// Run Station(s) (define when each needs to run)
fbStationINHeatAndSteam(
	aVehiclesStationFIFO:= aVehiclesStationFIFO,
	stReservation:= fbTrack.P_stReservation,
	stModeStateIn:= Input.Station.Station1.ModeState, 
	stModeStateOut := Output.Station.Station1.ModeState,
	bVehicleReadyAtInput:= eSeq <> E_VehicleOnStation.Idle, 
	bVehicleReadyAtOutput:= , 
	nCellStateCmd:= DINT_TO_UINT(eCommand),
	stJobDataIn:= Input.Station.Station1.JobData,  
	stConfigIn:= Input.Station.Station1.CurrentConfiguration, 
	stUpcomingConfigIn:= Input.Station.Station1.UpcomingConfiguration, 
	stControlIn := Input.Station.Station1.Control,
	stAdditionalDataIn := Input.Station.Station1.AdditionalData,
	sDistanceInDevice := Input.Transport.Configuration.Stations[2].StationLocation1.Position - Input.Transport.Configuration.Stations[1].StationLocation1.Position,
	stVehicleDataStaion := fbTrack.P_stVehicleDataOnStation,
	stJobDataOut := Output.Station.Station1.JobData,  
	stOEE := Output.Station.Station1.OEE, 
	stErrorWarning := Output.Station.Station1.ErrorWarning, 
	stConfigOut := Output.Station.Station1.CurrentConfiguration,
	stUpcomingConfigOut := Output.Station.Station1.UpcomingConfiguration,
	stOperationalDataOut := Output.Station.Station1.OperationalData, 
	stSustainabilityData := Output.Station.Station1.SustainabilityData, 
	stAdditionalDataOut := Output.Station.Station1.AdditionalData 	);
	
fbStationOUTHeatAndSteam(
	stModeStateIn:= Input.Station.Station2.ModeState, 
	stModeStateOut := Output.Station.Station2.ModeState,
	bVehicleReadyAtInput:= , 
	bVehicleReadyAtOutput:= , 
	nCellStateCmd:= DINT_TO_UINT(eCommand),
	stJobDataIn:= Input.Station.Station2.JobData,  
	stConfigIn:= Input.Station.Station2.CurrentConfiguration, 
	stUpcomingConfigIn:= Input.Station.Station2.UpcomingConfiguration, 
	stControlIn := Input.Station.Station2.Control,
	stAdditionalDataIn := Input.Station.Station1.AdditionalData,
	stJobDataOut := Output.Station.Station2.JobData,  
	stOEE := Output.Station.Station2.OEE, 
	stErrorWarning := Output.Station.Station2.ErrorWarning, 
	stConfigOut := Output.Station.Station2.CurrentConfiguration,
	stUpcomingConfigOut := Output.Station.Station2.UpcomingConfiguration,
	stOperationalDataOut := Output.Station.Station2.OperationalData, 
	stSustainabilityData := Output.Station.Station2.SustainabilityData, 
	stAdditionalDataOut := Output.Station.Station2.AdditionalData 	);

	
// Run Track Client
fbTrack(bEnable := , // Enabled in State Resetting
		bEStopOK := TRUE,
		bSuspend := , 
		bReset:= , 
		stCommand:= Input.Transport.Command,
		stMappingIn:= input.Transport.Mapping,
		stAdditionalDataIn:= Input.Transport.AdditionalData,
		bConnectedMethod=> , 
		bBusyMethod=> , 
		bConnectedNode=> , 
		bErrorMethod=> , 
		nErrorMethodID=> , 
		bErrorNode=> , 
		nErrorNodeID=> , 
		stStatus := Output.Transport.Status,
		stMappingOut := Output.Transport.Mapping, 
		stAdditionaldataOut := Output.Transport.AdditionalData,
		bStarted=> , 
		bSuspended=> 	);


//Set Station ready for vehicle to track
fbTrack.P_StationEmptyReady := eSeq = E_VehicleOnStation.Idle;
//fbTrack.P_bStationReady:=fbStationINHeatAndSteam.bStationReadyIn;

//Vehicles on station FIFO handling
M_VehicleOnStation(iCarrierCount=>diVehiclesInDevice);


//Set station empty for track - for vehicles going straight through
fbTrack.P_bStationEmpty:= diVehiclesInDevice = 0;

//Set FIFO for Station IN and Track Client
//fbStationINHeatAndSteam.P_CarriersFIFO := aVehiclesStationFIFO;
fbTrack.P_CarriersFIFO := aVehiclesStationFIFO;
END_METHOD

METHOD PROTECTED M_ErrorWarning
VAR_INPUT
END_VAR
VAR
	iAlNo				: UINT;
	iNoOfAlarms			: UINT;
	iNoOfWarnings		: UINT;
	bST1ErrWarDataChange: BOOL;
	bST2ErrWarDataChange: BOOL;
	bCellDataChange		: BOOL;
	bTCErrWarDataChange	: BOOL;
END_VAR
//Alarm / Warnings Cell
//bCellDataChange S= 
//M_ErrorWarningObj(arErrorWaringData:= arErrorWarningDataCell,
//	bActive:= eLineCtrl_EStop <> E_TwinSAFE_Logic_State.RUN, 
//	iErrorWarningType:= 2, 
//	diErrorWarningID:= E_AlarmCategory.Safety + 0, 
//	sDeviceID:= 'Global Safety',
//	iSeverity:= 2, 
//	iNativeID:= 0, 
//	sNativeMessage:= 'Emergency stop Line Controller');

//bCellDataChange S= 
//M_ErrorWarningObj(arErrorWaringData:= arErrorWarningDataCell,
//	bActive:= NOT bEStop_OK, 
//	iErrorWarningType:= 2, 
//	diErrorWarningID:= E_AlarmCategory.Safety + 20, 
//	sDeviceID:= 'Local Safety',
//	iSeverity:= 2, 
//	iNativeID:= 0, 
//	sNativeMessage:= 'Emergency stop Cell');

//bCellDataChange S= 
//M_ErrorWarningObj(arErrorWaringData:= arErrorWarningDataCell,
//	bActive:= eSHL_F70 <> E_TwinSAFE_Logic_State.RUN, 
//	iErrorWarningType:= 2, 
//	diErrorWarningID:= E_AlarmCategory.Safety + 21, 
//	sDeviceID:= 'Local Safety',
//	iSeverity:= 2, 
//	iNativeID:= 0, 
//	sNativeMessage:= 'Emergency stop Robot');
	
//bCellDataChange S= 
//M_ErrorWarningObj(arErrorWaringData:= arErrorWarningDataCell,
//	bActive:= NOT bDoor_OK, 
//	iErrorWarningType:= 2, 
//	diErrorWarningID:= E_AlarmCategory.Safety + 22, 
//	sDeviceID:= 'Local Safety',
//	iSeverity:= 2, 
//	iNativeID:= 0, 
//	sNativeMessage:= 'Cell Door 1 Not OK');
	
//bCellDataChange S= 
//M_ErrorWarningObj(arErrorWaringData:= arErrorWarningDataCell,
//	bActive:= stStatusData.e03_11_AK01_M3011 = E_Cylinder_Sta.Cyl_Sta_Err, 
//	iErrorWarningType:= 2, 
//	diErrorWarningID:= E_AlarmCategory.LifterStation1Device + 0, 
//	sDeviceID:= 'Lifter Station 1',
//	iSeverity:= 2, 
//	iNativeID:= 0, 
//	sNativeMessage:= 'Error Radial Gripper');
	
//bCellDataChange S= 
//M_ErrorWarningObj(arErrorWaringData:= arErrorWarningDataCell,
//	bActive:= stStatusData.e03_11_AK01_M3015 = E_Cylinder_Sta.Cyl_Sta_Err, 
//	iErrorWarningType:= 2, 
//	diErrorWarningID:= E_AlarmCategory.LifterStation1Device + 1, 
//	sDeviceID:= 'Lifter Station 1',
//	iSeverity:= 2, 
//	iNativeID:= 0, 
//	sNativeMessage:= 'Error Lifter Cylinder');
	
//bCellDataChange S= 
//M_ErrorWarningObj(arErrorWaringData:= arErrorWarningDataCell,
//	bActive:= stStatusData.e03_11_AK01_M3111 = E_Cylinder_Sta.Cyl_Sta_Err, 
//	iErrorWarningType:= 2, 
//	diErrorWarningID:= E_AlarmCategory.LifterStation2Device + 0, 
//	sDeviceID:= 'Lifter Station 2',
//	iSeverity:= 2, 
//	iNativeID:= 0, 
//	sNativeMessage:= 'Error Radial Gripper');
	
//bCellDataChange S= 
//M_ErrorWarningObj(arErrorWaringData:= arErrorWarningDataCell,
//	bActive:= stStatusData.e03_11_AK01_M3115 = E_Cylinder_Sta.Cyl_Sta_Err, 
//	iErrorWarningType:= 2, 
//	diErrorWarningID:= E_AlarmCategory.LifterStation2Device + 1, 
//	sDeviceID:= 'Lifter Station 2',
//	iSeverity:= 2, 
//	iNativeID:= 0, 
//	sNativeMessage:= 'Error Lifter Cylinder');

	
(*------------------------------------------------------------------------------------------------*)	
	
//Update alarm / warning list output to OPC
bST1ErrWarDataChange := iST1ErrWarDataChange <> Output.Station.Station1.ErrorWarning.DataChange;
iST1ErrWarDataChange := Output.Station.Station1.ErrorWarning.DataChange;
bST2ErrWarDataChange := iST2ErrWarDataChange <> Output.Station.Station2.ErrorWarning.DataChange;
iST2ErrWarDataChange := Output.Station.Station2.ErrorWarning.DataChange;
bTCErrWarDataChange := iTCErrWarDataChange <> fbTrack.stErrorWarning.DataChange;
iTCErrWarDataChange := fbTrack.stErrorWarning.DataChange;

IF bST1ErrWarDataChange OR bTCErrWarDataChange OR bCellDataChange THEN
	//Clear alarm list
	M_ErrorWarningClear();

	//Add alarm/warnings for Cell
	M_ErrorWarningAdd(arInErrorWarningList:= arErrorWarningDataCell, sLocationID:= 'C000004');
	
	//Add alarm/warnings for Station 1
	M_ErrorWarningAdd(arInErrorWarningList:= Output.Station.Station1.ErrorWarning.ErrorWarningData, sLocationID:= 'S000003');
	
	//Add alarm/warnings for Station 2
	M_ErrorWarningAdd(arInErrorWarningList:= Output.Station.Station2.ErrorWarning.ErrorWarningData, sLocationID:= 'S00000C');
	
	//Add alarm/warnings for Track Client
	M_ErrorWarningAdd(arInErrorWarningList:= fbTrack.stErrorWarning.ErrorWarningData, sLocationID:= 'TrackClient');
	
	stErrorWarning.DataChange := stErrorWarning.DataChange +1;
	//Output.Cell.ErrorWarning := stErrorWarning;
END_IF
END_METHOD

{attribute 'object_name' := 'M_Execute'}
METHOD M_Execute

IF (output.Station.Station1.ModeState.CurrentState = E_PML_State.Holding) THEN
	bHoldLocal := TRUE;
ELSIF (output.Station.Station1.ModeState.CurrentState = E_PML_State.Suspending) THEN
	bSuspendLocal := TRUE;
ELSIF (output.Station.Station1.ModeState.CurrentState <> E_PML_State.Execute) THEN
	// Exit execute state when all station(s) are not executing
	
	M_StateComplete();
END_IF
END_METHOD

{attribute 'object_name' := 'M_Held'}
METHOD M_Held
END_METHOD

{attribute 'object_name' := 'M_Holding'}
METHOD M_Holding

(*
// Check station(s) state
IF (fbBrushing.stOutput.stModeState.iCurrentState = E_PML_State.Held) THEN
	M_StateComplete();
END_IF
*)

// Do not wait for station state
//eCommand := E_PML_Command.Undefined;
M_StateComplete();
END_METHOD

{attribute 'object_name' := 'M_Idle'}
METHOD M_Idle
END_METHOD

METHOD PROTECTED M_Init : BOOL
VAR_INPUT
END_VAR

VAR
	SerialNumber: INT;
END_VAR

(*
	TEST OF ONLINE CHANGES WITH MERGE BRANCHES
*)
(*
	TEST OF ONLINE CHANGES WITH MERGE BRANCHES
*)
(*
	TEST OF ONLINE CHANGES WITH MERGE BRANCHES
*)
IF (NOT bInitDone) THEN
	// Set init done to TRUE. Set to false during init if needed
	bInitDone := TRUE;
	
// Track Client setup
	fbTrack.P_eCellType := E_CellType.Type_Inline;
	fbTrack.P_sCellID := 'C000004';
	fbTrack.P_sTrackserverURL := GVL.sVars.sTrackserver;
	fbTrack.P_sTrackserverNetID := GVL.sVars.sTrackserver_AMS;
	fbTrack.P_nTrackserverPort := 851;
	//Next station on track
	//fbTrack.P_sNextStationOnTrack := 'S000001';	// Cell 5
	fbTrack.P_sNextStationOnTrack := 'MMDP1C000000';	// Cell 5
	// Paths
	
	// Station(s)
	bInitDone := bInitDone AND
	fbTrack.M_DefineStation(nStationNo := 1,
							sStationID := Input.Transport.Configuration.Stations[1].StationID,							//S000003
							nLoc1PathID := Input.Transport.Configuration.Stations[1].StationLocation1.Path,				//17
							rLoc1Position := Input.Transport.Configuration.Stations[1].StationLocation1.Position,		//1.000
							nLoc2PathID := 0, //Input.Transport.Configuration.Stations[1].StationLocation2.Path,
							rLoc2Position := 0, //Input.Transport.Configuration.Stations[1].StationLocation2.Position,
							nLocDecPathID := Input.Transport.Configuration.DecisionPointLocation.Path,					//17
							rLocDecPosition := Input.Transport.Configuration.DecisionPointLocation.Position,			//0.650
							nPreBufferSize := 0, //Input.Transport.Configuration.Stations[1].PreBufferSize,
							nPostBufferSize := 0); //Input.Transport.Configuration.Stations[1].PostBufferSize );
							
		fbTrack.M_DefineStation(nStationNo := 2,
							sStationID := Input.Transport.Configuration.Stations[2].StationID,							//S00000C
							nLoc1PathID := Input.Transport.Configuration.Stations[2].StationLocation1.Path,				//17
							rLoc1Position := Input.Transport.Configuration.Stations[2].StationLocation1.Position,		//1.850
							nLoc2PathID := 0, //Input.Transport.Configuration.Stations[2].StationLocation2.Path,
							rLoc2Position := 0, //Input.Transport.Configuration.Stations[2].StationLocation2.Position,
							nLocDecPathID := Input.Transport.Configuration.DecisionPointLocation.Path,					//17
							rLocDecPosition := Input.Transport.Configuration.DecisionPointLocation.Position,			//0.650
							nPreBufferSize := 0, //Input.Transport.Configuration.Stations[2].PreBufferSize,
							nPostBufferSize := 0); //Input.Transport.Configuration.Stations[2].PostBufferSize );
	
	// Cell information
	Output.Header.CellInformation.CellID := 'C000004';
	Output.Header.CellInformation.CellName := 'Cell 4';
	Output.Header.CellInformation.NumberOfStations := 2;
	Output.Header.MetaInformation.CellType := 'Inline';
	Output.Header.MetaInformation.InterfaceVersion := 0;
	Output.Header.MetaInformation.PLCVersion := nPLCVersion;
	Output.Header.MetaInformation.SerialNumber := sSerialIPC;
	
	// Station information
	Output.Header.CellInformation.StationInformation[1].NumberOfOperations := 1;
	Output.Header.CellInformation.StationInformation[1].StationID := 'S000003';
	Output.Header.CellInformation.StationInformation[1].StationName := 'HeatAndSteam In';
	Output.Station.Station1.CurrentConfiguration.OP11600.ToolCapacity := 0;
	Output.Station.Station1.CurrentConfiguration.OP11600.MaterialCapacity := 0;
	
	Output.Header.CellInformation.StationInformation[2].NumberOfOperations := 0;
	Output.Header.CellInformation.StationInformation[2].StationID := 'S00000C';
	Output.Header.CellInformation.StationInformation[2].StationName := 'HeatAndSteam Out';
//	Output.Station.Station2.CurrentConfiguration.OP11601.ToolCapacity := 0;
//	Output.Station.Station2.CurrentConfiguration.OP11601.MaterialCapacity := 0;

	
	// Operation information
	Output.Header.CellInformation.StationInformation[1].OperationInformation[1].OperationID := 'OP11600';
	Output.Header.CellInformation.StationInformation[1].OperationInformation[1].OperationName := 'HeatAndSteam Step 1';
	
	// Transport information
	Output.Header.CellInformation.TransportInformation.TransportName := 'C000004';
	Output.Header.CellInformation.TransportInformation.TransportType := 'Inline';
	
	// Components
	
	//Specify Sustainability data
	Output.Cell.SustainabilityData.Energy[1] := F_NewDeviceDataX(	'HS', 						'Heat and Steam', 
																	E_AlarmCategory.OP11600 +0, 	'Instant Power', 				E_Units._KW);
END_IF
END_METHOD

METHOD PROTECTED M_OEEHandling
VAR_INPUT
END_VAR
VAR
	bChanged			: BOOL;
END_VAR
// Call base FB method
SUPER^.M_OEEHandling();


// Product counters
IF ( stOEE.ProcessedProduct <> (Output.Station.Station1.OEE.ProcessedProduct) ) THEN
	stOEE.ProcessedProduct := Output.Station.Station1.OEE.ProcessedProduct;
	bChanged := TRUE;
END_IF
IF ( stOEE.GoodProduct <> (Output.Station.Station1.OEE.GoodProduct) ) THEN
	stOEE.GoodProduct := Output.Station.Station1.OEE.GoodProduct;
	bChanged := TRUE;
END_IF
IF ( stOEE.RejectedProduct <> (Output.Station.Station1.OEE.RejectedProduct) ) THEN
	stOEE.RejectedProduct := Output.Station.Station1.OEE.RejectedProduct;
	bChanged := TRUE;
END_IF

// Update Event ID!
// TODO!!!
stOEE.EventID;

// Increment DataChange to signal to LC that sometihng has changed
IF (bChanged) THEN
	// Update time for changes
	stOEE.DateTime := SYSTEMTIME_TO_DT(TIMESTR := fbGetTime.TIMESTR);
	
	stOEE.DataChange := stOEE.DataChange + 1;
END_IF
END_METHOD

{attribute 'object_name' := 'M_Resetting'}
METHOD M_Resetting
VAR
	bDone : BOOL;
END_VAR
// Track
fbTrack.bEnable := TRUE;

IF (fbTrack.bStarted AND fbTrack.bTrackInitDone AND fbTrack.bVehicleInitDone) OR bBypassTrack THEN
	eCommand := E_PML_Command.Undefined;
	M_StateComplete();
	bBypassTrack := FALSE;
END_IF
END_METHOD

{attribute 'object_name' := 'M_Starting'}
METHOD M_Starting
(*
// Check station(s)
IF (fbBrushing.stModeStateOut.CurrentState = E_PML_State.Execute) THEN
	bStartLocal := FALSE;
	M_StateComplete();
END_IF
*)

eCommand := E_PML_Command.Undefined;
M_StateComplete();
END_METHOD

{attribute 'object_name' := 'M_Stopped'}
METHOD M_Stopped
END_METHOD

{attribute 'object_name' := 'M_Stopping'}
METHOD M_Stopping
//eCommand := E_PML_Command.Undefined;
M_StateComplete();
END_METHOD

{attribute 'object_name' := 'M_Suspended'}
METHOD M_Suspended
END_METHOD

{attribute 'object_name' := 'M_Suspending'}
METHOD M_Suspending
//fbTrack.bSuspend := TRUE;

// Check station(s) state
//IF ( (output.Station.Station1.ModeState.CurrentState = E_PML_State.Suspended) AND fbTrack.bSuspended ) THEN
//	eCommand := E_PML_Command.Undefined;
	M_StateComplete();
//END_IF
END_METHOD

METHOD M_SustainabilityDataHandling
VAR_INPUT
END_VAR
Output.Cell.SustainabilityData.Energy[1].Value := Output.Station.Station1.OperationalData.OP11600.DeviceData[4].Value;
END_METHOD

{attribute 'object_name' := 'M_Undefined'}
METHOD M_Undefined
END_METHOD

{attribute 'object_name' := 'M_Unholding'}
METHOD M_Unholding

// Check station(s) state
IF ((output.Station.Station1.ModeState.CurrentState  <> E_PML_State.Held)) THEN
//	eCommand := E_PML_Command.Undefined;
	M_StateComplete();
END_IF
END_METHOD

{attribute 'object_name' := 'M_Unsuspending'}
METHOD M_Unsuspending
//eCommand := E_PML_Command.Undefined;
fbTrack.bSuspend := FALSE;
M_StateComplete();
(*
// Check station(s) state
IF (fbBrushing.stModeStateOut.CurrentState <> E_PML_State.Suspended) THEN
	M_StateComplete();
END_IF
*)
END_METHOD

METHOD M_VehicleOnStation : BOOL
VAR_INPUT
END_VAR
VAR
	bVehiclePresent			: BOOL;
	iCarrierIndex			: UINT;
	iCarrierID				: STRING;
	i						: UINT;
	j						: UINT;
	fPositionOut			: REAL;
	sTempString				: STRING(200);
END_VAR
VAR_OUTPUT
	iCarrierCount			: UINT;
END_VAR
//Carrier count
iCarrierCount := 0;
FOR i := 1 TO 10 DO
	IF (aVehiclesStationFIFO[i].sCarrierID = '') THEN
		EXIT;//End reached
	ELSE
		iCarrierCount := iCarrierCount + 1;
	END_IF 
END_FOR

CASE eSeq OF
	E_VehicleOnStation.Idle:
		IF fbTrack.bReadyStationIn[1] THEN
			stVehicleDataOnStation := fbTrack.P_stVehicleDataOnStation; //Read out vehicle data to temp
			eSeq := E_VehicleOnStation.VehicleAtStation;
			F_LogFile(CONCAT('Cell Vehicle On Station - New Vehicle station IN, Veh NO: ', TO_STRING(stVehicleDataOnStation.stVehicle.nVehicleID)));
		END_IF
		
	E_VehicleOnStation.VehicleAtStation:
		tonSeqTimer(IN := TRUE, PT := T#10S);
		IF output.Station.Station1.ModeState.CurrentState = E_PML_State.Starting (*AND NOT fbStationINHeatAndSteam.P_bSkipVehicle*) THEN
			tonSeqTimer(IN := FALSE);
			eSeq := E_VehicleOnStation.AddToFIFO;
			F_LogFile(CONCAT('Cell Vehicle On Station - Vehicle at station, Veh NO: ', TO_STRING(stVehicleDataOnStation.stVehicle.nVehicleID)));
//		ELSIF fbStationINHeatAndSteam.P_bSkipVehicle THEN
//			tonSeqTimer(IN := FALSE);
//			eSeq := E_VehicleOnStation.WaitStationStart;
//			F_LogFile(CONCAT('Cell Vehicle On Station - Vehicle at station SKIPPED, Veh NO: ', TO_STRING(stVehicleDataOnStation.stVehicle.nVehicleID)));
		END_IF
		
		// Check if vehicle is waiting for station start or skip
		IF (tonSeqTimer.Q) THEN
			// Force update of vehicle status to OPC/Line Controller
			tonSeqTimer(IN := FALSE);
			fbTrack.P_bForceVehicleUpdateOPC := TRUE;
		END_IF
		
	E_VehicleOnStation.AddToFIFO:
		
		FOR i := 1 TO 10 DO
			IF (aVehiclesStationFIFO[i].sCarrierID = '') THEN
				aVehiclesStationFIFO[i].sCarrierID := stVehicleDataOnStation.stVehicle.sCarrierID;
				aVehiclesStationFIFO[i].nVehicleNo := stVehicleDataOnStation.stVehicle.nVehicleID;
				aVehiclesStationFIFO[i].JobData := Output.Station.Station1.JobData.OP11600;
				aVehiclesStationFIFO[i].fVelocity := fbStationINHeatAndSteam.fVelocityCal;
				
				sTempString := CONCAT('Station FIFO - Carrier with ID: ', TO_STRING(aVehiclesStationFIFO[i].sCarrierID));
				sTempString := CONCAT(sTempString, ' added to FIFO, Vehicle no: ');
				sTempString := CONCAT(sTempString, TO_STRING(aVehiclesStationFIFO[i].nVehicleNo));
				sTempString := CONCAT(sTempString, ', Velocity: ');
				F_LogFIle(CONCAT(sTempString, TO_STRING(aVehiclesStationFIFO[i].fVelocity)));
				
				EXIT;
			END_IF
		END_FOR
		
		eSeq := E_VehicleOnStation.WaitStationStart;
		F_LogFile(CONCAT('Cell Vehicle On Station - Add FIFO, Veh NO: ', TO_STRING(stVehicleDataOnStation.stVehicle.nVehicleID)));
		
	E_VehicleOnStation.WaitStationStart:
	
		IF output.Station.Station1.ModeState.CurrentState = E_PML_State.Completing THEN
			//fbStationINHeatAndSteam.P_bSkipVehicle := FALSE;
			eSeq := E_VehicleOnStation.MoveVehicle;
			F_LogFile(CONCAT('Cell Vehicle On Station - Station completing, Veh NO: ', TO_STRING(stVehicleDataOnStation.stVehicle.nVehicleID)));
		END_IF
		
	E_VehicleOnStation.MoveVehicle:
		IF (fbStationINHeatAndSteam.P_bSkipVehicle) THEN
			// Set vehicle velocity to 1 if skipped!
			iRes := fbTrack.M_CallMoveVehicleToStationIn(	eInputType := E_MMVehicleInputType.eMMVehicleInputType_VehicleID, 
															sInput := UINT_TO_STRING(stVehicleDataOnStation.stVehicle.nVehicleID), 
															sStationID := fbTrack.aStations[2].sStationID,//'S00000C',
															eDirection := E_MMDirection.eMMDirection_Forward, 
															fVelocity := 1.0, 
															fAcceleration := 1	);
		ELSE
			iRes := fbTrack.M_CallMoveVehicleToStationIn(	eInputType := E_MMVehicleInputType.eMMVehicleInputType_VehicleID, 
															sInput := UINT_TO_STRING(stVehicleDataOnStation.stVehicle.nVehicleID), 
															sStationID := fbTrack.aStations[2].sStationID,//'S00000C',
															eDirection := E_MMDirection.eMMDirection_Forward, 
															fVelocity := fbStationINHeatAndSteam.fVelocityCal, 
															fAcceleration := 1	);
		END_IF

		IF (iRes = 2) THEN
			// Movement call OK
			fbTrack.P_bVehicleMovedFromSt1 := TRUE;
			eSeq := E_VehicleOnStation.VehicleLeftStation;
			
			sTempString := CONCAT('Cell Vehicle On Station - Vehicle No: ', TO_STRING(stVehicleDataOnStation.stVehicle.nVehicleID));
			sTempString := CONCAT(sTempString, ' Move OK towards station 2, with velocity: ');
			F_LogFIle(CONCAT(sTempString, TO_STRING(fbStationINHeatAndSteam.fVelocityCal)));
		ELSIF (iRes = 3) THEN
			// Movement call failed
			eSeq := E_VehicleOnStation.VehicleLeftStation;
			
			sTempString := CONCAT('Cell Vehicle On Station - Vehicle No: ', TO_STRING(stVehicleDataOnStation.stVehicle.nVehicleID));
			sTempString := CONCAT(sTempString, ' Move FAILED towards station 2, with velocity: ');
			F_LogFIle(CONCAT(sTempString, TO_STRING(fbStationINHeatAndSteam.fVelocityCal)));
		END_IF
	
	E_VehicleOnStation.VehicleLeftStation:
		eSeq := E_VehicleOnStation.Idle;
		
		F_LogFile(CONCAT('Cell Vehicle - Vehicle left station, Veh NO: ', TO_STRING(stVehicleDataOnStation.stVehicle.nVehicleID)));
END_CASE

//Remove from FIFO
IF fbTrack.P_iVehicleFifoOut > 0 THEN
	FOR i := 1 TO 9 DO
		IF aVehiclesStationFIFO[i].nVehicleNo = fbTrack.P_iVehicleFifoOut THEN
			sTempString := CONCAT('Cell VehicleOnStat: Vehicle#: ', TO_STRING(aVehiclesStationFIFO[1].nVehicleNo));
			fbTrack.M_VehicleToReadRemove(aVehiclesStationFIFO[1].nVehicleNo);
			sTempString := CONCAT(sTempString, ' Removed from FIFO place: ');
			F_LogFile(CONCAT(sTempString, TO_STRING(i)));
			
			aVehiclesStationFIFO[i] := aDummyVehicleStationData;
		END_IF
	END_FOR
	fbTrack.P_iVehicleFifoOut := 0;
END_IF
//IF fbTrack.P_bFifoOut THEN
	
//	IF (aVehiclesStationFIFO[1].sCarrierID <> '') THEN
//		sTempString := CONCAT('Station FIFO - FIFO out carrierID: ', TO_STRING(aVehiclesStationFIFO[1].sCarrierID));
//		fbTrack.M_VehicleToReadRemove(aVehiclesStationFIFO[1].nVehicleNo);
//		F_LogFIle(CONCAT(sTempString, ' Removed from FIFO'));
//	END_IF
		
//	aVehiclesStationFIFO[1].sCarrierID := '';
//	aVehiclesStationFIFO[1].fCalculatedTIA := 0.0;
//	aVehiclesStationFIFO[1].fVelocity := 0.0;
//	aVehiclesStationFIFO[1].nVehicleNo := 0;
//	fbTrack.P_bFifoOut := FALSE;
//END_IF


//Clean up FIFO
FOR i := 1 TO 9 DO
//	IF LEN(aVehiclesStationFIFO[i].sCarrierID) = 0 AND LEN(aVehiclesStationFIFO[i+1].sCarrierID) <> 0 THEN
	IF (aVehiclesStationFIFO[i].sCarrierID = '') AND (aVehiclesStationFIFO[i+1].sCarrierID <> '') THEN 
		aVehiclesStationFIFO[i] := aVehiclesStationFIFO[i+1]; // Move next item here
		aVehiclesStationFIFO[i+1] := aDummyVehicleStationData;
	END_IF
END_FOR	

//Update estimated time to reach station 2
tonVehicleDataRead(IN := TRUE, PT := T#1S);	// Read vehicle data every second
fPositionOut := Input.Transport.Configuration.Stations[2].StationLocation1.Position;
FOR i := 1 TO 10 DO
	IF (aVehiclesStationFIFO[i].sCarrierID = '') THEN
		EXIT;
	END_IF //End reached
	
	// Trig vehicle data reading
	IF (tonVehicleDataRead.Q) THEN
		fbTrack.M_VehicleToReadAdd(aVehiclesStationFIFO[i].nVehicleNo);
	END_IF
	
	FOR j := 1 TO 1000 DO
		IF (Output.Transport.Status.Carrier[i].CarrierID = '') THEN
			EXIT;
		END_IF //End reached
		
		IF (aVehiclesStationFIFO[i].sCarrierID = Output.Transport.Status.Carrier[j].CarrierID) THEN
			IF (aVehiclesStationFIFO[i].fVelocity > 0.001) THEN
				// Calculate remaining time for reaching station 2 location using remaining distance and commanded velocity
				aVehiclesStationFIFO[i].fCalculatedTIA := (Input.Transport.Configuration.Stations[2].StationLocation1.Position - Output.Transport.Status.Carrier[j].CurrentPosition) / aVehiclesStationFIFO[i].fVelocity;
			END_IF
		END_IF
	END_FOR
END_FOR
// Timer for reading vehicle data for vehicles in the FIFO buffer
IF (tonVehicleDataRead.Q) THEN
	tonVehicleDataRead(IN := FALSE);
END_IF

//Set empty out
M_VehicleOnStation := iCarrierCount = 0;

//Cyclic log FIFO timer
IF iCarrierCount > 0 THEN
	diFifoLogTimer := diFifoLogTimer + g_iPLCScan_MS;
	IF diFifoLogTimer > 10000 THEN
		FOR i := 1 TO iCarrierCount DO
			sTempString := CONCAT('Station FIFO - Status, Carrier ID: ', TO_STRING(aVehiclesStationFIFO[i].sCarrierID));
			sTempString := CONCAT(sTempString, ', Vehicle no: ');
			sTempString := CONCAT(sTempString, TO_STRING(aVehiclesStationFIFO[i].nVehicleNo));
			sTempString := CONCAT(sTempString, ', Velocity: ');
			sTempString := CONCAT(sTempString, TO_STRING(aVehiclesStationFIFO[i].fVelocity));
			sTempString := CONCAT(sTempString, ', TIA: ');
			F_LogFIle(CONCAT(sTempString, TO_STRING(aVehiclesStationFIFO[i].fCalculatedTIA)));
		END_FOR
		diFifoLogTimer := 0;
	END_IF
END_IF
END_METHOD

END_FUNCTION_BLOCK

// ---- ECC/Basic/Cell/FB_Cell_Basic.TcPOU
/// Generic FB for cells/stations
/// Contains the PackML state machine and PackTags data
FUNCTION_BLOCK FB_Cell_Basic EXTENDS FB_PLC_Basic IMPLEMENTS ITF_UnitState 
VAR_INPUT
	bResetEStop				: BOOL;
	bLockDoor				: BOOL;
	bUnlockDoor				: BOOL;
	bCellLight				: BOOL;
	iHeartBeatFromMES		: UINT;
END_VAR
VAR_OUTPUT
	bModeChangeInProcess	: BOOL;
	bEStopOK				: BOOL;						// Will result in Abort state in PackML!
	bDoorsOK				: BOOL;
	bCellLightOn			: BOOL;
	iHeartBeatToMES			: UINT;

	bUndefinedDone			: BOOL;						// When the SPS is started, the first state is Undefiend. bUndefinedDone is TRUE, when the method Undefined has succesful finished
	bInvalidModeCommandOut	: BOOL;
	bChangeIntoProduction	: BOOL;
	bStationCommError		: BOOL := FALSE;			// Error communication with station PLC/HW
END_VAR
VAR_IN_OUT
	stModeStateIn			: ST_InputModeState;
	stModeStateOut			: ST_OutputModeState;
	stOEE					: ST_OutputOEE;
	stErrorWarning			: ST_OutputErrorWarning;
END_VAR
VAR
// Mode and State requests
	// Input:
	eMode					: E_PMLProtectedUnitMode := E_PMLProtectedUnitMode.ePMLProtUnitMode_Production;
	eCommand				: E_PMLCommand := E_PMLCommand.ePMLCommand_Undefined;
	bModeChangeRequest		: BOOL;
	// Output:
	eRequestedMode			: E_PMLProtectedUnitMode;
	eCurrentMode			: E_PMLProtectedUnitMode;
	eRequestedState			: E_PMLState;
	eCurrentState			: E_PMLState;	
	
// PackML
	fbUnitModeManager		: PML_UnitModeManager;		// The PML_UnitModeManager manage the Modechanges
	fbStateMachine 			: PML_StateMachine;			// The PML_StateMachine mangae the Statechanges
	nStateModeChange		: INT	:= 0;				// Variable to handle the modechange
	nLastState				: E_PMLState;				// Variable to store last state
	bProductionLocal		: BOOL := FALSE;			// Local Production mode button/command. Must be updated in inherited FB's
	bManualLocal			: BOOL := FALSE;			// Local Manual mode button/command. Must be updated in inherited FB's
	bMaintenanceLocal		: BOOL := FALSE;			// Local Maintenance mode button/command. Must be updated in inherited FB's
	bAbortLocal				: BOOL := FALSE;			// Local abort button/command. Must be updated in inherited FB's
	bStartLocal				: BOOL := FALSE;			// Local start button/command. Must be updated in inherited FB's
	bStopLocal				: BOOL := FALSE;			// Local stop button/command. Must be updated in inherited FB's
	bResetLocal				: BOOL := FALSE;			// Local reset button/command. Must be updated in inherited FB's
	bClearLocal				: BOOL := FALSE;			// Local clear button/command. Must be updated in inherited FB's
	bHoldLocal				: BOOL := FALSE;			// Local hold button/command. Must be updated in inherited FB's
	bUnholdLocal			: BOOL := FALSE;			// Local unhold button/command. Must be updated in inherited FB's
	bSuspendLocal			: BOOL := FALSE;			// Local hold button/command. Must be updated in inherited FB's
	bUnsuspendLocal			: BOOL := FALSE;			// Local unhold button/command. Must be updated in inherited FB's
//Error warning
	arErrorWarningDataCell	: ARRAY [1..255] OF ST_ErrorWarningDataX;
// Recipe	
//	fbRecipe				: FB_RecipeData;			// Recipe data
// DateTime
	fbGetTimePML			: FB_GetTimePML;
// HeartBeat
	fbHeartBeatGen			: FB_GenerateHeartBeat;
	fbHeartBeatCheck		: FB_CheckHeartBeat;
// Misc
	fbGetTime				: NT_GetTime;
END_VAR
VAR_IN_OUT
//	stCommand				: ST_PMLc_ECC;
//	stStatus				: ST_PMLs_ECC;
//	stAdmin					: ST_PMLa_ECC;
//	stService				: ST_PMLse_ECC;
END_VAR
VAR PERSISTENT
	sLineCtrlNetID	AT %Q*	: AMSNETID := [10,38,190,120,1,1];
	iCellID			AT %Q*	: UINT;
END_VAR

// Run parent FB!
SUPER^();

// Get system time
fbGetTime(	NETID:= '',	// Local PLC 
			START:= NOT fbGetTime.START AND NOT fbGetTime.BUSY, 
			TMOUT:= T#5S	);

// Heart beat
fbHeartBeatGen(iHeartBeat => iHeartBeatToMES);
fbHeartBeatCheck(iHeartBeat := iHeartBeatFromMES);		

// OEE
M_OEEHandling();			

// Mode state handshake handling
IF ((stModeStateIn.ChangeRequest <> stModeStateOut.ChangeStatus) AND (stModeStateIn.ChangeRequest > 0)) THEN
	// Mode change
	IF ( (stModeStateIn.Mode > 0) AND (stModeStateIn.Mode <= 6) ) THEN
		// Set acknowledge
		IF (stModeStateOut.ChangeAcknowledge <> stModeStateIn.ChangeRequest) THEN
			stModeStateOut.ChangeAcknowledge := stModeStateIn.ChangeRequest;
			stModeStateOut.ModeStateResponse := 0;
			stModeStateOut.DataChange := stModeStateOut.DataChange + 1;
		END_IF
		// Set new mode
		eMode := stModeStateIn.Mode;
		stModeStateOut.RequestedMode := DINT_TO_UINT(eMode);
		// Wait done
		IF (stModeStateIn.Mode = eCurrentMode) THEN
			// Set change status
			stModeStateOut.ChangeStatus := stModeStateIn.ChangeRequest;
			stModeStateOut.ModeStateResponse := 3;
			stModeStateOut.DataChange := stModeStateOut.DataChange + 1;
			stModeStateIn.Mode := E_PML_Mode.Undefined;
		END_IF
	END_IF

	// State change
	IF ( (stModeStateIn.State > 0) AND (stModeStateIn.State <= 10) ) THEN
		// Set acknowledge
		IF (stModeStateOut.ChangeAcknowledge <> stModeStateIn.ChangeRequest) THEN
			stModeStateOut.ChangeAcknowledge := stModeStateIn.ChangeRequest;
			stModeStateOut.ModeStateResponse := 0;
			stModeStateOut.DataChange := stModeStateOut.DataChange + 1;
		END_IF
		// Set new state command
		eCommand := stModeStateIn.State;
		CASE eCommand OF
			E_PML_Command.Reset:
				stModeStateOut.RequestedState := E_PML_State.Idle;

			E_PML_Command.Start:
				stModeStateOut.RequestedState := E_PML_State.Execute;
			
			E_PML_Command.Stop:
				stModeStateOut.RequestedState := E_PML_State.Stopped;
			
			E_PML_Command.Hold:
				stModeStateOut.RequestedState := E_PML_State.Held;
			
			E_PML_Command.Unhold:
				stModeStateOut.RequestedState := E_PML_State.Execute;
			
			E_PML_Command.Suspend:
				stModeStateOut.RequestedState := E_PML_State.Suspended;
			
			E_PML_Command.Unsuspend:
				stModeStateOut.RequestedState := E_PML_State.Execute;
			
			E_PML_Command.Abort:
				stModeStateOut.RequestedState := E_PML_State.Aborted;
			
			E_PML_Command.Clear:
				stModeStateOut.RequestedState := E_PML_State.Stopped;
			
			E_PML_Command.Complete:
				stModeStateOut.RequestedState := E_PML_State.Complete;
			
		END_CASE
		// Wait done
		IF (stModeStateOut.RequestedState = eCurrentState) THEN
			// Set change status
			stModeStateOut.ChangeStatus := stModeStateIn.ChangeRequest;
			stModeStateOut.DataChange := stModeStateOut.DataChange + 1;
			stModeStateOut.ModeStateResponse := 3;
			stModeStateIn.State := E_PML_Command.Undefined;
			eCommand := E_PML_Command.Undefined;
		END_IF
	END_IF
END_IF

// Run State Machine
M_PackML_StateMachine();


// Update current mode/state
IF (DINT_TO_UINT(eCurrentMode) <> stModeStateOut.CurrentMode) THEN
	stModeStateOut.CurrentMode := DINT_TO_UINT(eCurrentMode);
	stModeStateOut.DataChange := stModeStateOut.DataChange + 1;	
END_IF
IF (DINT_TO_UINT(eCurrentState) <> stModeStateOut.CurrentState) THEN
	stModeStateOut.CurrentState := DINT_TO_UINT(eCurrentState);
	stModeStateOut.DataChange := stModeStateOut.DataChange + 1;	
END_IF

/// Static state "Aborted"
/// Trigged by "StateCompleted" when in "Aborting" state
/// Requires "Clear" to go to "Clearing" state 
{attribute 'object_name' := 'M_Aborted'}
METHOD M_Aborted
END_METHOD

/// Dynamic state "Aborting"
/// Trigged by "Abort" command
/// Requires "StateCompleted" to go to "Aborted" state 
{attribute 'object_name' := 'M_Aborting'}
METHOD M_Aborting
M_StateComplete();
END_METHOD

/// Dynamic state "Clearing"
/// Trigged by "Clear" command "Aborted" state
/// Requires "StateCompleted" to go to "Stopped" state 
{attribute 'object_name' := 'M_Clearing'}
METHOD M_Clearing
M_StateComplete();
END_METHOD

/// Static state "Complete"
/// Trigged by "StateCompleted" when in "Completing" state
/// Requires "Reset" to go to "Resetting" state 
{attribute 'object_name' := 'M_Complete'}
METHOD M_Complete
END_METHOD

/// Dynamic state "Completing"
/// Trigged by "StageCompleted" command when in "Execute" state
/// Requires "StateCompleted" to go to "Complete" state 
{attribute 'object_name' := 'M_Completing'}
METHOD M_Completing
M_StateComplete();
END_METHOD

METHOD M_ErrorWarningAdd : BOOL
VAR_INPUT
	//stInErrorWarning: ST_OutputErrorWarning;
	
	sLocationID		: STRING;
END_VAR
VAR_IN_OUT
	arInErrorWarningList: ARRAY [1..255] OF ST_ErrorWarningDataX;
END_VAR
VAR
	i				: UINT;
	j				: UINT:=1;
	iNoAlarms		: UINT;
	iNoWarnings		: UINT;
END_VAR
FOR i:= 1 TO 255 DO
	IF arInErrorWarningList[i].ErrorWarningID <> 0 THEN
		REPEAT
			//Find first empty spot
			IF stErrorWarning.ErrorWarningData[j].ErrorWarningID = 0 THEN
				
				stErrorWarning.ErrorWarningData[j] := arInErrorWarningList[i];
				stErrorWarning.ErrorWarningData[j].LocationID := sLocationID;
				
				IF stErrorWarning.ErrorWarningData[j].ErrorWarningType = 1 THEN
					iNoWarnings := iNoWarnings +1;
				ELSIF stErrorWarning.ErrorWarningData[j].ErrorWarningType = 2 THEN
					iNoAlarms := iNoAlarms +1;
				END_IF
				
				EXIT;
			END_IF
			j := j + 1;
		UNTIL j = 255 END_REPEAT
	ELSE
		EXIT;
	END_IF
END_FOR

//Update number of erros and warnings
stErrorWarning.NumberOfErrors := stErrorWarning.NumberOfErrors + iNoAlarms;
stErrorWarning.NumberOfWarnings := stErrorWarning.NumberOfWarnings + iNoWarnings;
END_METHOD

METHOD M_ErrorWarningClear : BOOL
VAR_INPUT

END_VAR
VAR
	i				: UINT;
END_VAR
//FOR i:= 1 TO 255 DO
//	MEMSET(ADR(stErrorWarning.ErrorWarningData[i]), 0, SIZEOF(stErrorWarning.ErrorWarningData[i]));
//END_FOR
MEMSET(ADR(stErrorWarning.ErrorWarningData), 0, SIZEOF(stErrorWarning.ErrorWarningData));

stErrorWarning.NumberOfErrors := 0;
stErrorWarning.NumberOfWarnings := 0;
END_METHOD

METHOD M_ErrorWarningObj : BOOL
VAR_INPUT
	bActive				: BOOL;
	iErrorWarningType	: UINT;
	diErrorWarningID 	: UDINT;
	sDeviceID			: STRING(30);
	iSeverity			: UINT;
	iNativeID			: UDINT;
	sNativeMessage		: STRING(80);
END_VAR
VAR_IN_OUT
	arErrorWaringData	: ARRAY [1..255] OF ST_ErrorWarningDataX;
END_VAR
VAR
	iFoundPos			: UINT;
	i					: UINT;
	j					: UINT;
END_VAR
//Look through array to find existing record(s)
FOR i := 1 TO 255 DO
	IF arErrorWaringData[i].ErrorWarningID = 0 THEN
		EXIT;
	END_IF
	//Existing alarm - first
	IF arErrorWaringData[i].ErrorWarningID = diErrorWarningID AND iFoundPos = 0 THEN
		iFoundPos := i;
	//Multiple records - delete
	ELSIF arErrorWaringData[i].ErrorWarningID = diErrorWarningID AND iFoundPos <> 0 THEN
		MEMSET(ADR(arErrorWaringData[i]), 0, SIZEOF(arErrorWaringData[i]));
		M_ErrorWarningObj := TRUE;
	END_IF
END_FOR

//Alarm high
IF bActive THEN
	//New alarm
	IF iFoundPos = 0 THEN
		arErrorWaringData[i].ErrorWarningType := iErrorWarningType;
		arErrorWaringData[i].DeviceID := sDeviceID;
		arErrorWaringData[i].Severity := iSeverity;
		arErrorWaringData[i].NativeID := iNativeID;
		arErrorWaringData[i].NativeMessage := sNativeMessage;
		arErrorWaringData[i].ErrorWarningID := diErrorWarningID;
		arErrorWaringData[i].DateTime := SYSTEMTIME_TO_STRING(fbGetTime.TIMESTR);
		M_ErrorWarningObj := TRUE;
	END_IF
	
//Alarm low
ELSIF NOT bActive AND iFoundPos <> 0 THEN
	MEMSET(ADR(arErrorWaringData[iFoundPos]), 0, SIZEOF(arErrorWaringData[iFoundPos]));
	M_ErrorWarningObj := TRUE;
END_IF

//Defrag
IF M_ErrorWarningObj THEN
	FOR i:= 1 TO 254 DO
		//Find first empty spot
		IF arErrorWaringData[i].ErrorWarningID = 0 THEN
			//Find first record
			FOR j:= i TO 255 DO
				IF arErrorWaringData[j].ErrorWarningID <> 0 THEN
					//Move to empty spot
					arErrorWaringData[i] := arErrorWaringData[j];
					MEMSET(ADR(arErrorWaringData[j]), 0, SIZEOF(arErrorWaringData[j]));
					EXIT;
				END_IF
			END_FOR
		END_IF
		//No more records
		IF j >= 255 THEN
			RETURN;
		END_IF
	END_FOR
END_IF
END_METHOD

/// Static state "Execute"
/// Trigged by "StageCompleted" when in "Starting" state
/// Trigged by "StageCompleted" when in "Unholding" state
/// Trigged by "StageCompleted" when in "Unsuspending" state
/// Requires "Hold" command to go to "Holding" state 
/// Requires "Suspend" command to go to "Suspending" state 
/// Requires "StageCompleted" to go to "Completing" state 
{attribute 'object_name' := 'M_Execute'}
METHOD M_Execute
M_StateComplete();
END_METHOD

/// Static state "Held"
/// Trigged by "StateCompleted" when in "Holding" state
/// Requires "Unhold" command to go to "Unholding" state 
{attribute 'object_name' := 'M_Held'}
METHOD M_Held
END_METHOD

/// Dynamic state "Holding"
/// Trigged by "Hold" command when in "Execute" state
/// Requires "StateCompleted" to go to "Held" state 
{attribute 'object_name' := 'M_Holding'}
METHOD M_Holding
M_StateComplete();
END_METHOD

/// Static state "Idle"
/// Trigged by "StateCompleted" when in "Resetting" state
/// Requires "Start" command to go to "Starting" state 
{attribute 'object_name' := 'M_Idle'}
METHOD M_Idle
END_METHOD

METHOD PROTECTED M_OEEHandling
VAR_INPUT
END_VAR
// Must be overloaded in derived FB's!
;
END_METHOD

METHOD PROTECTED M_PackML_StateMachine : BOOL
VAR_INPUT
END_VAR

CASE nStateModeChange OF

	0:	// Waiting for user request
		IF (NOT bModeChangeInProcess) THEN
			// Local unit mode change request
			IF (bProductionLocal AND (eCurrentMode <> Tc3_PackML_V2.ePMLProtUnitMode_Production)) THEN
				eMode := ePMLProtUnitMode_Production;
				bModeChangeRequest := TRUE;
			ELSIF (bManualLocal AND (eCurrentMode <> Tc3_PackML_V2.ePMLProtUnitMode_Manual)) THEN
				eMode := ePMLProtUnitMode_Manual;
				bModeChangeRequest := TRUE;
			ELSIF (bMaintenanceLocal AND (eCurrentMode <> Tc3_PackML_V2.ePMLProtUnitMode_Maintenance)) THEN
				eMode := ePMLProtUnitMode_Maintenance;
				bModeChangeRequest := TRUE;
			END_IF
		END_IF
		bChangeIntoProduction := FALSE;
		IF ((eMode = ePMLProtUnitMode_Production) AND (eCurrentMode = ePMLProtUnitMode_Invalid)) THEN
			nStateModeChange := 1;
		ELSIF (bModeChangeRequest AND (eMode <> ePMLProtUnitMode_Production)) THEN
			nStateModeChange := 1;
		ELSIF ((eMode = ePMLProtUnitMode_Production) AND (eCurrentMode <> ePMLProtUnitMode_Production)) THEN
			nStateModeChange := 3;
		END_IF
		
	1:	// Starting UnitModeManager 
		fbUnitModeManager.bExecute := TRUE;
		fbUnitModeManager.eModeCommand := eMode;
		bModeChangeInProcess := TRUE;
	
		IF (fbUnitModeManager.bDone) THEN
			fbUnitModeManager.bExecute := FALSE;
			bInvalidModeCommandOut := FALSE;
			nStateModeChange := 0;
			bChangeIntoProduction := FALSE;
			bModeChangeInProcess := FALSE;
		ELSIF (fbUnitModeManager.bError) THEN
			bInvalidModeCommandOut := TRUE;
			fbUnitModeManager.bExecute := FALSE;
			nLastState := eCurrentState;
			nStateModeChange := 2;
			bChangeIntoProduction := FALSE;
			bModeChangeInProcess := FALSE;
		END_IF
	
	2:	// ErrorHanddling
		IF (bModeChangeRequest) THEN
			nStateModeChange := 0;
			bInvalidModeCommandOut := FALSE;
		ELSIF (nLastState <> eCurrentState) THEN
			bInvalidModeCommandOut := FALSE;
		END_IF
		
	3:	// state to check, if command 'Production' is valid
		IF ((eCurrentState = ePMLState_Aborted) OR (eCurrentState = ePMLState_Stopped) OR (eCurrentState = ePMLState_Idle)) THEN
			bChangeIntoProduction := TRUE;
			nStateModeChange := 1;
		ELSE
			nStateModeChange := 2;
			bInvalidModeCommandOut := TRUE;
			nLastState := eCurrentState;
		END_IF
END_CASE


// Run Unit Mode Manager
fbUnitModeManager(	eState := eCurrentState,
					eModeStatus => eCurrentMode,
					bDone => ,
					bError => ,
					nErrorId => 	);

IF (fbUnitModeManager.eModeStatus <> 0) THEN
	// Local E-stop/abort handling	
	IF (NOT bEStopOK OR bAbortLocal) THEN
		eCommand := E_PMLCommand.ePMLCommand_Abort;
	// Local Start handling
	ELSIF (bStartLocal) THEN
		eCommand := E_PMLCommand.ePMLCommand_Start;
	// Local Stop handling
	ELSIF (bStopLocal) THEN
		eCommand := E_PMLCommand.ePMLCommand_Stop;
	// Local Reset handling
	ELSIF (bResetLocal) THEN
		eCommand := E_PMLCommand.ePMLCommand_Reset;
	// Local Clear handling
	ELSIF (bClearLocal) THEN
		eCommand := E_PMLCommand.ePMLCommand_Clear;
	// Local Hold handling
	ELSIF (bHoldLocal) THEN
		eCommand := E_PMLCommand.ePMLCommand_Hold;
	// Local Unhold handling
	ELSIF (bUnholdLocal) THEN
		eCommand := E_PMLCommand.ePMLCommand_Unhold;
	// Local Suspend handling
	ELSIF (bSuspendLocal) THEN
		eCommand := E_PMLCommand.ePMLCommand_Suspend;
	// Local Unsuspend handling
	ELSIF (bSuspendLocal) THEN
		eCommand := E_PMLCommand.ePMLCommand_Unsuspend;
	// 
	ELSIF (stModeStateIn.State = 0) THEN
		eCommand := E_PMLCommand.ePMLCommand_Undefined;
	END_IF
	
	// Calling the StateMachine, when there is a valid Mode
	fbStateMachine(	eMode := eCurrentMode, 				
					eCommand := eCommand,			
					stSubUnitInfoRef := ,
					stOptions := , 
					eState => eCurrentState, 				
					bError => , 
					nErrorID => 	);

END_IF

// Requested state:
CASE eCommand OF			
	E_PMLCommand.ePMLCommand_Abort:
		eRequestedState := E_PMLState.ePMLState_Aborted;
		
	E_PMLCommand.ePMLCommand_Clear:
		eRequestedState := E_PMLState.ePMLState_Stopped;

	E_PMLCommand.ePMLCommand_Complete:
		eRequestedState := E_PMLState.ePMLState_Complete;
		
	E_PMLCommand.ePMLCommand_Hold:
		eRequestedState := E_PMLState.ePMLState_Held;
		
	E_PMLCommand.ePMLCommand_Reset:
		eRequestedState := E_PMLState.ePMLState_Idle;
		
	E_PMLCommand.ePMLCommand_Start:
		eRequestedState := E_PMLState.ePMLState_Execute;
		
	E_PMLCommand.ePMLCommand_Stop:
		eRequestedState := E_PMLState.ePMLState_Stopped;
		
	E_PMLCommand.ePMLCommand_Suspend:
		eRequestedState := E_PMLState.ePMLState_Suspended;
		
	E_PMLCommand.ePMLCommand_Unhold:
		eRequestedState := E_PMLState.ePMLState_Execute;
		
	E_PMLCommand.ePMLCommand_Unsuspend:
		eRequestedState := E_PMLState.ePMLState_Execute;
		
END_CASE

//One of the methods is executing by the actual state
CASE eCurrentState OF
	ePMLState_Undefined:
		M_Undefined();
	ePMLState_Clearing:
		M_Clearing();
	ePMLState_Stopped:
		M_Stopped();
	ePMLState_Starting:
		M_Starting();
	ePMLState_Idle:
		M_Idle();
	ePMLState_Suspended:
		M_Suspended();
	ePMLState_Execute:
		M_Execute();
	ePMLState_Stopping:
		M_Stopping();
	ePMLState_Aborting:
		M_Aborting();
	ePMLState_Aborted:
		M_Aborted();
	ePMLState_Holding:
		M_Holding();
	ePMLState_Held:
		M_Held();
	ePMLState_Unholding:
		M_Unholding();
	ePMLState_Suspending:
		M_Suspending();
	ePMLState_Unsuspending:
		M_Unsuspending();
	ePMLState_Resetting:
		M_Resetting();
	ePMLState_Completing:
		M_Completing();
	ePMLState_Complete:
		M_Complete();
END_CASE
END_METHOD

/// Dynamic state "Resetting"
/// Trigged by "Reset" command when in "Stopped" state
/// Requires "StateCompleted" to go to "Idle" state 
{attribute 'object_name' := 'M_Resetting'}
METHOD M_Resetting
M_StateComplete();
END_METHOD

/// Dynamic state "Starting"
/// Trigged by "Start" command when in "Idle" state
/// Requires "StateCompleted" to go to "Execute" state 
{attribute 'object_name' := 'M_Starting'}
METHOD M_Starting
M_StateComplete();
END_METHOD

{attribute 'object_name' := 'M_StateComplete'}
METHOD M_StateComplete
//the actual state is completed
fbStateMachine.M_StateComplete();
END_METHOD

/// Static state "Stopped"
/// Trigged by "StateCompleted" when in "Stopping" state
/// Requires "Reset" command to go to "Resetting" state 
{attribute 'object_name' := 'M_Stopped'}
METHOD M_Stopped
END_METHOD

/// Dynamic state "Stopping"
/// Trigged by "Stop" command
/// Requires "StateCompleted" to go to "Stopped" state 
{attribute 'object_name' := 'M_Stopping'}
METHOD M_Stopping
M_StateComplete();
END_METHOD

/// Static state "Suspended"
/// Trigged by "StateCompleted" when in "Suspending" state
/// Requires "Unsuspend" command to go to "Unsuspending" state 
{attribute 'object_name' := 'M_Suspended'}
METHOD M_Suspended
END_METHOD

/// Dynamic state "Suspending"
/// Trigged by "Suspend" command when in "Execute" state
/// Requires "StateCompleted" to go to "Suspended" state 
{attribute 'object_name' := 'M_Suspending'}
METHOD M_Suspending
M_StateComplete();
END_METHOD

{attribute 'object_name' := 'M_Undefined'}
METHOD M_Undefined
END_METHOD

/// Dynamic state "Unholding"
/// Trigged by "Unhold" command when in "Held" state
/// Requires "StateCompleted" to go to "Execute" state 
{attribute 'object_name' := 'M_Unholding'}
METHOD M_Unholding
M_StateComplete();
END_METHOD

/// Dynamic state "Unsuspending"
/// Trigged by "Unsuspend" command when in "Suspended" state
/// Requires "StateCompleted" to go to "Execute" state 
{attribute 'object_name' := 'M_Unsuspending'}
METHOD M_Unsuspending
M_StateComplete();
END_METHOD

END_FUNCTION_BLOCK

// ---- ECC/Basic/Cell/FB_PLC_Basic.TcPOU
/// Generic FB for all ECC PLC's
FUNCTION_BLOCK FB_PLC_Basic
VAR_INPUT
END_VAR
VAR_OUTPUT
	rCPUTemp				: REAL;
	rSafetyTemp				: REAL;
	sSerialIPC				: STRING;					// IPC serial number
	sSerialMB				: STRING;					// Mainboard serial number
	rCPULoadPLC				: REAL;						// CPU load for the PLC runtime
	rCPULoad				: REAL;						// CPU load for the system
	rCPUFrequency			: REAL;						// CPU frequency	
END_VAR
VAR
// HW
	License_State	AT %I*	: WORD := 8;	// State from Ethercat module
	License_AdsAdrr	AT %I*	: AMSADDR;		// ADS address from EtherCAT module
// Persistent data
	fbPersistentData		: Tc2_SUPS.FB_S_UPS_CX51x0;
	bUPS_PowerFailDetected	: BOOL;
	eUPS_State				: Tc2_SUPS.E_S_UPS_State;
// Misc
	fbCPUTemp				: FB_GetCPUTemp;			// CPU temp
	fbSafetyTemp			: FB_GetSafetyTemp;			// Safety CPU temp
	fbIPCSerial				: FB_GetIPCSerial;			// IPC serial number
	bGetIPCSerial			: BOOL := TRUE;				// 
	fbCPULoadPLC			: FB_GetCPULoadPLC;			// Get actual CPU load (for the PLC runtime !)
	fbCPULoad				: FB_GetCPULoad;			// Get actual CPU load (for system !)
END_VAR


// Persistent data
fbPersistentData(	sNetID:= '', 			// Local PLC
					iPLCPort:= 851, 		// PLC runtime #1
					iUPSPort:= 16#588,
					tTimeout:= T#5S, 
					eUpsMode:= E_S_UPS_Mode.eSUPS_WrPersistData_Shutdown, 
					ePersistentMode:= E_PersistentMode.SPDM_2PASS, 
					tRecoverTime:= T#10S, 
					bPowerFailDetect=> bUPS_PowerFailDetected, 
					eState=> eUPS_State);

// Get CPU temp
fbCPUTemp(	rInterval := 10,	// [s]
			rCPUTemp => rCPUTemp,
			bError => ,
			nErrID => );

// Get Safety Temp
fbSafetyTemp(	rInterval := 10,	// [s]
				rSafetyTemp => rSafetyTemp,
				bError => ,
				nErrID =>	);

// Get serials
fbIPCSerial(bExecute := bGetIPCSerial,
			sSerialIPC => sSerialIPC,
			sSerialMainBoard => sSerialMB,
			bError => ,
			nErrID => 	);
bGetIPCSerial := FALSE;

// Get CPU load for PLC runtime
fbCPULoadPLC(	rInterval := 2,
				rCPULoad => rCPULoadPLC,
				bError => ,
				nErrID => 	);

// Get CPU load for System
fbCPULoad(	rInterval := 2,
			rCPULoad => rCPULoad,
			rCPUFrequency => rCPUFrequency,
			bError => ,
			nErrID => 	);

// PLC scan time
IF (g_rPLCScan_S <= 0.0) THEN
	g_rPLCScan_S := UDINT_TO_LREAL(_TaskInfo[GETCURTASKINDEXEX()].CycleTime) / 10000000.0;
	g_iPLCScan_MS := UDINT_TO_UINT(_TaskInfo[GETCURTASKINDEXEX()].CycleTime / 10000);
END_IF

END_FUNCTION_BLOCK

// ---- ECC/Tools/FB_GetCPUTemp.TcPOU
FUNCTION_BLOCK FB_GetCPUTemp
VAR_INPUT
	rInterval			: REAL := 10.0;		// [sec]
END_VAR
VAR_OUTPUT
	rCPUTemp			: REAL;				// [deg]
	bError				: BOOL;				// error flag (indicator: error occured)
	nErrID				: UDINT;			// last error ID 
END_VAR
VAR
	// internal use
	sAmsNetId			: STRING := '';		// ADS Net ID (local = '')    
	iState				: INT;
	uData				: UINT;
	stMDP_Addr			: Tc2_MDP.ST_MDP_Addr;
	// FB instances
	fbReadMDPElement	: Tc2_MDP.FB_MDP_ReadElement;  
	tonInterval			: Tc2_Standard.TON;
END_VAR


// Interval timer
tonInterval(IN := NOT tonInterval.Q, PT := REAL_TO_TIME(rInterval * 1000.0));

CASE iState OF
	0: // Initiate program parameters (if required)
		fbReadMDPElement(bExecute := FALSE);
		IF (tonInterval.Q) THEN
			iState := 10;
		END_IF

	10:	// Trigger FB: request CPU data
		stMDP_Addr.nArea := INT_TO_BYTE(Tc2_MDP.eMDP_Area_ConfigArea);
		stMDP_Addr.nTableId := 1;
		stMDP_Addr.nSubIdx := 3;
		fbReadMDPElement(	bExecute := TRUE,
							eModuleType := Tc2_MDP.eMDP_ModT_CPU,
							stMDP_Addr := stMDP_Addr,
							iModIdx := 0,
							pDstBuf := ADR(uData),
							cbDstBufLen := SIZEOF(uData),
							sAmsNetId := sAmsNetId	);
		iState := 20;

	20:	// Process FB: Request CPU temp
		fbReadMDPElement(bExecute := FALSE); 
		IF (NOT fbReadMDPElement.bBusy) THEN
			IF (fbReadMDPElement.bError) THEN
				bError := TRUE;
				nErrID := fbReadMDPElement.nErrID; 
				iState := 0;
			ELSE
				bError := FALSE;
				rCPUTemp := UINT_TO_REAL(uData);
				iState := 30;
			END_IF                                               
		END_IF
    
     30: // Done 
		iState := 0;

	ELSE
		iState := 0; 

END_CASE

END_FUNCTION_BLOCK

// ---- ECC/Tools/FB_GetSafetyTemp.TcPOU
FUNCTION_BLOCK FB_GetSafetyTemp
VAR_INPUT
	rInterval			: REAL := 10.0;		// [sec]
END_VAR
VAR_OUTPUT
	rSafetyTemp			: REAL;				// [deg]
	bError				: BOOL;				// error flag (indicator: error occured)
	nErrID				: UDINT;			// last error ID 
END_VAR
VAR
	tonInterval			: Tc2_Standard.TON;
	fbSafetyTemp		: TC2_EtherCAT.FB_EcCoESdoRead;
	sSafetyNetID AT %I*	: AMSADDR;			// Map to Safety module 'AdsAddr'
	iSafetyTemp			: INT;
END_VAR


// Interval timer
tonInterval(IN := NOT tonInterval.Q, PT := REAL_TO_TIME(rInterval * 1000.0));

// Read value
fbSafetyTemp(	sNetId:= F_CreateAmsNetId(sSafetyNetID.netId), 
				nSlaveAddr:= sSafetyNetID.port, 
				nIndex:= 16#F984, 	// Device Info Data C1
				nSubIndex:= 16#2, 	// Temperature C1
				pDstBuf:= ADR(iSafetyTemp), 
				cbBufLen:= SIZEOF(iSafetyTemp), 
				bExecute:= tonInterval.Q, 
				tTimeout:= T#5S,  
				bBusy=> , 
				bError=> bError, 
				nErrId=> nErrID	);

// scale output
rSafetyTemp := INT_TO_REAL(iSafetyTemp);

END_FUNCTION_BLOCK

// ---- ECC/Tools/FB_GetIPCSerial.TcPOU
FUNCTION_BLOCK FB_GetIPCSerial
VAR_INPUT
	bExecute			: BOOL;				// TRUE to start
END_VAR
VAR_OUTPUT
	sSerialIPC			: STRING;			// Serial no of IPC
	sSerialMainBoard	: STRING;			// Serial no of Mainboard
	bError				: BOOL;				// error flag (indicator: error occured)
	nErrID				: UDINT;			// last error ID 
END_VAR
VAR
	// internal use
	sAmsNetId			: STRING := '';		// ADS Net ID (local = '')    
	iState				: INT;
	sData				: STRING;
	stMDP_Addr			: Tc2_MDP.ST_MDP_Addr;
	// FB instances
	fbReadMDPElement	: Tc2_MDP.FB_MDP_ReadElement;  
	fbReadMDPIndex		: Tc2_MDP.FB_MDP_ReadIndex;
END_VAR


CASE iState OF
	0: // Initiate program parameters (if required)
		fbReadMDPElement(bExecute := FALSE);
		fbReadMDPIndex(bExecute := FALSE);
		IF (bExecute) THEN
			iState := 10;
		END_IF

	10:	// Trigger FB: request mainboard data
		sData := '';
		stMDP_Addr.nArea := INT_TO_BYTE(Tc2_MDP.eMDP_Area_ConfigArea);
		stMDP_Addr.nTableId := 1;
		stMDP_Addr.nSubIdx := 2;
		fbReadMDPElement(	bExecute := TRUE,
							eModuleType := Tc2_MDP.eMDP_ModT_Mainboard,
							stMDP_Addr := stMDP_Addr,
							iModIdx := 0,
							pDstBuf := ADR(sData),
							cbDstBufLen := SIZEOF(sData),
							sAmsNetId := sAmsNetId	);
		iState := 20;

	20:	// Process FB: Request mainboard serial
		fbReadMDPElement(bExecute := FALSE); 
		IF (NOT fbReadMDPElement.bBusy) THEN
			IF (fbReadMDPElement.bError) THEN
				bError := TRUE;
				nErrID := fbReadMDPElement.nErrID; 
				iState := 0;
			ELSE
				bError := FALSE;
				sSerialMainBoard := sData;
				iState := 30;
			END_IF                                               
		END_IF
  
	30:	// trigger FB: request single index in MDP Device Area, IPC serial number
		sData           := '';
		fbReadMDPIndex(	bExecute := TRUE,
						nIndex := 16#F9F0,
						nSubIndex := 0,
						pDstBuf := ADR(sData),
						cbDstBufLen := SIZEOF(sData),
						sAmsNetId := sAmsNetId 	);
		iState := 40;
            
	40:	// Process FB: request single index in MDP Device Area, IPC serial number
		fbReadMDPIndex(bExecute := FALSE); 
		IF (NOT fbReadMDPIndex.bBusy) THEN
			IF (fbReadMDPIndex.bError) THEN
				bError := TRUE;
				nErrID := fbReadMDPIndex.nErrID; 
			ELSE
				bError := FALSE;
				sSerialIPC := sData;
			END_IF
			iState := 90;
		END_IF		
  
     90: // Done
		IF (NOT bExecute) THEN
			iState := 0;
		END_IF

	ELSE
		iState := 0; 

END_CASE

END_FUNCTION_BLOCK

// ---- ECC/Tools/FB_GetCPULoadPLC.TcPOU
FUNCTION_BLOCK FB_GetCPULoadPLC
VAR_INPUT
	rInterval			: REAL := 10.0;		// [sec]
END_VAR
VAR_OUTPUT
	rCPULoad			: REAL;				// [deg]
	bError				: BOOL;				// error flag (indicator: error occured)
	nErrID				: UDINT;			// last error ID 
END_VAR
VAR
	// internal use
	sAmsNetId			: T_AmsNetId;		// ADS Net ID (local = '')    
	iState				: INT;
	// FB instances
	fbReadCPUUsage		: TC_CpuUsage;  
	tonInterval			: Tc2_Standard.TON;
	// Info
	iErrorCnt			: UINT;
	iGoodCnt			: UINT;
END_VAR


// Interval timer
tonInterval(IN := NOT tonInterval.Q, PT := REAL_TO_TIME(rInterval * 1000.0));

CASE iState OF
	0: // Initiate program parameters (if required)
		fbReadCPUUsage(START := FALSE);
		IF (tonInterval.Q) THEN
			iState := 10;
		END_IF

	10:	// Trigger FB: request CPU data
		fbReadCPUUsage(	NETID := sAmsNetId,
						START := TRUE,
						TMOUT := T#5S	);
		IF (fbReadCPUUsage.BUSY) THEN
			// Started
			iState := 20;
		ELSIF (fbReadCPUUsage.ERR) THEN
			// Error
			iErrorCnt := iErrorCnt + 1;
			iState := 0;
		END_IF

	20:	// Process FB: Request CPU temp
		fbReadCPUUsage(START := FALSE); 
		IF (NOT fbReadCPUUsage.BUSY) THEN
			IF (NOT fbReadCPUUsage.ERR) THEN
				rCPULoad := fbReadCPUUsage.USAGE;
				iGoodCnt := iGoodCnt + 1;
				iState := 30;
			ELSE
				iErrorCnt := iErrorCnt + 1;
				iState := 0;
			END_IF                                               
		END_IF
    
     30: // Done 
		iState := 0;

	ELSE
		iState := 0; 

END_CASE

bError := fbReadCPUUsage.ERR;
nErrID := fbReadCPUUsage.ERRID;

END_FUNCTION_BLOCK

// ---- ECC/Tools/FB_GetCPULoad.TcPOU
FUNCTION_BLOCK FB_GetCPULoad
VAR_INPUT
	rInterval			: REAL := 10.0;		// [sec]
END_VAR
VAR_OUTPUT
	rCPULoad			: REAL;				// [%]
	rCPUFrequency		: REAL;
	bError				: BOOL;				// error flag (indicator: error occured)
	nErrID				: UDINT;			// last error ID 
END_VAR
VAR
	// internal use
	sAmsNetId			: STRING := '';		// ADS Net ID (local = '')    
	iState				: INT;
	uData				: UINT;
    stMDP_ModuleHeader  : ST_MDP_ModuleHeader;
    stMDP_ModuleContent : ST_MDP_CPU;
	// FB instances
	fbReadMDPCPU		: Tc2_MDP.FB_MDP_CPU_Read;
	tonInterval			: Tc2_Standard.TON;
	// Info
	iErrorCnt			: UINT;
	iGoodCnt			: UINT;
END_VAR


// Interval timer
tonInterval(IN := NOT tonInterval.Q, PT := REAL_TO_TIME(rInterval * 1000.0));

CASE iState OF
	0: // Initiate program parameters (if required)
		fbReadMDPCPU(bExecute := FALSE);
		IF (tonInterval.Q) THEN
			iState := 10;
		END_IF

	10:	// Trigger FB: request CPU data
		fbReadMDPCPU(	bExecute := TRUE,
						tTimeout := T#5S,
						iModIdx := 0,
						sAmsNetId := sAmsNetId,
						stMDP_ModuleHeader => stMDP_ModuleHeader,
						stMDP_ModuleContent => stMDP_ModuleContent 	);
		iState := 20;

	20:	// Process FB: Request CPU temp
		fbReadMDPCPU(bExecute := FALSE); 
		IF (NOT fbReadMDPCPU.bBusy) THEN
			IF (fbReadMDPCPU.bError) THEN
				bError := TRUE;
				nErrID := fbReadMDPCPU.nErrID; 
				iErrorCnt := iErrorCnt + 1;
				iState := 0;
			ELSE
				bError := FALSE;
				rCPULoad := UINT_TO_REAL(stMDP_ModuleContent.iCPUusage);
				rCPUFrequency := UDINT_TO_REAL(stMDP_ModuleContent.iCPUfrequency);
				iGoodCnt := iGoodCnt + 1;
				iState := 30;
			END_IF                                               
		END_IF
    
     30: // Done 
		iState := 0;

	ELSE
		iState := 0; 

END_CASE

END_FUNCTION_BLOCK

// ---- ECC/Tools/FB_GetTimePML.TcPOU
FUNCTION_BLOCK FB_GetTimePML
VAR_INPUT
END_VAR
VAR_OUTPUT
	PML_Time		: ARRAY [0..6] OF DINT;
END_VAR
VAR
	fbGetTime		: NT_GetTime;
	tonInterval		: TON;
	tInterval		: TIME := T#100ms;
END_VAR


tonInterval(	IN := NOT tonInterval.Q,
				PT := tInterval,
				Q =>,
				ET =>	);

fbGetTime(	NETID:= '', 
			START:= tonInterval.Q, 
			TMOUT:= T#5S, 
			BUSY=> , 
			ERR=> , 
			ERRID=> , 
			TIMESTR=> 	);


PML_Time := TIMESTRUCT_TO_PackMLTime(fbGetTime.TIMESTR);

END_FUNCTION_BLOCK

// ---- ECC/Tools/FB_GenerateHeartBeat.TcPOU
FUNCTION_BLOCK FB_GenerateHeartBeat
VAR_INPUT
END_VAR
VAR_OUTPUT
	iHeartBeat		: UINT;
END_VAR
VAR
	tInterval		: TIME := T#500ms;
	tonInterval		: TON;
END_VAR


tonInterval(IN := TRUE,
			PT := tInterval,
			Q => );

IF (tonInterval.Q) THEN
	tonInterval(IN := FALSE);
	iHeartBeat := iHeartBeat + 1;
	IF (iHeartBeat > 100) THEN
		iHeartBeat := 0;
	END_IF
END_IF

PROPERTY PUBLIC P_tInterval : TIME
GET
P_tInterval := tInterval;
END_GET
SET
tInterval := P_tInterval;
END_SET
END_PROPERTY

END_FUNCTION_BLOCK

// ---- ECC/Tools/FB_CheckHeartBeat.TcPOU
FUNCTION_BLOCK FB_CheckHeartBeat
VAR_INPUT
	iHeartBeat		: UINT;
END_VAR
VAR_OUTPUT
	bOK				: BOOL;
END_VAR
VAR
	iHeartBeat_Old	: UINT;
	tofTimeOut		: TOF;
	tMaxTime		: TIME := T#500MS;
END_VAR


tofTimeOut(	IN := (iHeartBeat <> iHeartBeat_Old),
			PT := tMaxtime,
			Q => bOK);
iHeartBeat_Old := iHeartBeat;

PROPERTY PUBLIC P_tMaxTime : TIME
GET
P_tMaxTime := tMaxTime;
END_GET
SET
tMaxTime := P_tMaxTime;
END_SET
END_PROPERTY

END_FUNCTION_BLOCK

// ---- ECC/Cell_Unit_4/HeatAndSteam/FB_HeatAndSteamIN.TcPOU
FUNCTION_BLOCK FB_HeatAndSteamIN EXTENDS FB_Station_Basic
VAR_INPUT
	stReservation			: ST_ReservationData;		// Reservation on station
	sDistanceInDevice		: REAL;
	stVehicleDataStaion		: ST_ReadVehicleData ; //Data for vehicle on station in
END_VAR
VAR_OUTPUT
	fVelocityCal			: REAL;
	fTemperatureCal			: REAL;
	fSteamCal				: REAL;
	fAirCal					: REAL;
	fTimeCal				: REAL;
END_VAR
VAR_IN_OUT
	// Inputs
	stJobDataIn				: ST_InputStationHSJobData;
	stConfigIn				: ST_InputStationHSConfiguration;
	stUpcomingConfigIn		: ST_InputStationHSUpcomingConfiguration;
	stControlIn				: ST_InputStationHSControl;
	stAdditionalDataIn		: ST_InputStationHSAdditionalData;
	// Outputs
	stJobDataOut			: ST_OutputStationHSJobData;
	stConfigOut				: ST_OutputStationHSCurrentConfiguration;
	stUpcomingConfigOut		: ST_OutputStationHSUpcomingConfiguration;
	stOperationalDataOut	: ST_OutputStationHSOperationalData;
	stSustainabilityData	: ST_OutputStationHSSustainabilityData;
	stAdditionalDataOut		: ST_OutputStationHSAdditionalData;
	aVehiclesStationFIFO	: ARRAY[1..10] OF ST_VehicleInHS;
END_VAR 
VAR
	eSeq					: E_HSStationINSeq;
	eSeq_old				: E_HSStationINSeq;
	bStateChange_OS			: BOOL;
		
	fbHS_Driver				: FB_EMS_HS;
	stHSDriverWrite			: ST_EMS_HS_Write;
	stHSDriverRead			: ST_EMS_HS_Read;
	
	sWarningError			: ARRAY [1..21] OF STRING; // Delete when alarm section is agreed.
	bStationReadyIn			: BOOL;
	OperationOK				: BOOL;
	bTestActive				: BOOL;
	
	bSkipVehicle			: BOOL;
	iNextJobStation			: UINT;
	iNextJobStationOld		: UINT;
	

// Start up
	sCarrierID				: STRING; // Current carrier ID
	nCheckValid				: UINT;
	bTestBool				: BOOL;
	
	diStateTimer			: DINT;
	tonIdleTimer			: TON;
	i						: INT;
	iVehicleInFIFO			: UINT;
END_VAR

VAR CONSTANT
	
END_VAR

SUPER^( stModeStateIn := stModeStateIn,
		stModeStateOut := stModeStateOut,
		stOEE := stOEE,
		stErrorWarning := stErrorWarning);

		
IF bInitDone THEN
	M_ErrorWarning();
END_IF
		
M_Init();

//Automatic reset when operation complete
IF (eCommand <> ePMLCommand_Start AND eCurrentState = E_PMLState.ePMLState_Complete) THEN
	bResetLocal := TRUE;
END_IF

//Station in ready -> Cell -> TrackClient
//bStationReadyIn := eCurrentState = E_PMLState.ePMLState_Idle;

//Job Data
M_JobDataHandling();

//Line controller request
M_ConfigurationHandling();

//Device driver
M_DeviceDriver();

// Operational Data
M_OperationalDataHandling();

/// Static state "Aborted"
/// Trigged by "StateCompleted" when in "Aborting" state
/// Requires "Clear" to go to "Clearing" state 
{attribute 'object_name' := 'M_Aborted'}
METHOD M_Aborted
END_METHOD

/// Dynamic state "Aborting"
/// Trigged by "Abort" command
/// Requires "StateCompleted" to go to "Aborted" state 
{attribute 'object_name' := 'M_Aborting'}
METHOD M_Aborting
// Stop all moving parts
(* STOP all OPSTIONS and Track - Clear alarms og gå til Complete*)
eSeq := E_HSStationINSeq.Idle;

stHSDriverWrite.rSetFanSpeed := 0;
stHSDriverWrite.rSetTemp := 0;
stHSDriverWrite.stCommands.REMOTE_STOP := TRUE;
stHSDriverWrite.stCommands.REMOTE_START := FALSE;


M_StateComplete();
END_METHOD

(*Calculated velocity for needed operation

 TFinal=(TMachine∗cT+SMachine∗cS+AMachine∗cA)∗t+TInital
 TFinal = Final estimated upper temperature
 TMachine = Temperature of the heat radiation of the device
 SMachine = Steam level in the device
 AMachine = Air flow in the device
 TInitial = initial temperature of the upper
 t = Time upper spends in device
 cT = weighted factor transferring heat radiation to the upper temperature
 cS = weighted factor for the influence the steam level has to the upper temeperature
 cA = weighted factor for the influence the air flow has to the upper temeperature
*)
METHOD M_CalculatedVelocity : REAL
VAR_INPUT
	fTFinal			: REAL;
	fTInital		: REAL;
	fTMachine		: REAL;
	fSMachine		: REAL;
	fAMachine		: REAL;
	fcT				: REAL;
	fcS				: REAL;
	fcA				: REAL;
	fTravelLength	: REAL; //Length of travel from beginning to end of path
END_VAR
VAR
	fTimeSet		: REAL;
END_VAR
//Check settings
IF fcT = 0 THEN
	fcT := 0.0000059;
END_IF
IF fcS = 0 THEN
	fcS := 0.00000045;
END_IF
IF fcA = 0 THEN
	fcA := 0.000068;
END_IF


//Calculate time needed in device
//t = ( (TFinal) / (TMachine * cT + SMachine * cS + AMachine * cA) ) - TInitial
fTimeSet := (fTFinal - fTInital) / ((fTMachine * fcT) + (fSMachine * fcS) + (fAMachine * fcA));
//Velocity needed with current setting
M_CalculatedVelocity := fTravelLength/fTimeSet;

//Check velocity
IF M_CalculatedVelocity >= 0.001 AND M_CalculatedVelocity <= 2.0 THEN
	; //Ok
ELSE
	M_CalculatedVelocity := -1; // Not ok
END_IF
END_METHOD

METHOD M_ClearAll : BOOL
VAR_INPUT
END_VAR

IF eCurrentState = E_PMLState.ePMLState_Aborted THEN
	eSeq := E_HSStationINSeq.Idle;
	bSkipVehicle := FALSE;
	
	iNextJobStation := 0;
	iNextJobStationOLD := 0;
	
	F_Logfile('ST1 - All data cleared!');
	
	M_ClearAll := TRUE;
END_IF
END_METHOD

/// Dynamic state "Clearing"
/// Trigged by "Clear" command "Aborted" state
/// Requires "StateCompleted" to go to "Stopped" state 
{attribute 'object_name' := 'M_Clearing'}
METHOD M_Clearing
(* Clear all OPSTIONS and Track - Clear alarms og gå til Complete*)

M_StateComplete();
END_METHOD

/// Static state "Complete"
/// Trigged by "StateCompleted" when in "Completing" state
/// Requires "Reset" to go to "Resetting" state 
{attribute 'object_name' := 'M_Complete'}
METHOD M_Complete
END_METHOD

/// Dynamic state "Completing"
/// Trigged by "StageCompleted" command when in "Execute" state
/// Requires "StateCompleted" to go to "Complete" state 
{attribute 'object_name' := 'M_Completing'}
METHOD M_Completing

VAR
	
END_VAR



M_StateComplete();
END_METHOD

METHOD M_ConfigurationHandling
VAR_INPUT
END_VAR
VAR
	sTempSTring		: STRING(200);
END_VAR
// Is updated from operator/HMI
IF (stConfigIn.ChangeRequest <> stConfigOut.ChangeStatus) AND (stConfigIn.ChangeRequest > 0) THEN
	sTempString := CONCAT('ConfigChange request - Old request: ', TO_STRING(stConfigOut.ChangeStatus));
	sTempString := CONCAT(sTempString, ', New request: ');
	sTempString := CONCAT(sTempString, TO_STRING(stConfigIn.ChangeRequest));
	sTempString := CONCAT(sTempString, ' ConfigType: ');
	F_LogFile(CONCAT(sTempString, stConfigIn.ConfigurationType)); 
	
	// Change request from Line Controller
	IF (stAdditionalDataIn.MESHandShakes.DataChangeStatusCurrentConfiguration = stConfigOut.DataChange) THEN
		stConfigOut.ChangeAcknowledge := stConfigIn.ChangeRequest;
		stConfigOut.DataChange := stConfigOut.DataChange + 1;
	
		// Check Configuration Type
		IF (F_StringCompNoCase(stConfigIn.ConfigurationType, 'OP11600')) THEN	
			// Update output job data
			stConfigOut.ConfigurationType := stConfigIn.ConfigurationType;
			stConfigOut.DateTime := SYSTEMTIME_TO_DT(timestr:=fbGetTime.TIMESTR);
			stConfigOut.OP11600 := stConfigIn.OP11600;
			
			// Signal that job data has been written		
			stConfigOut.ChangeStatus := stConfigIn.ChangeRequest;
			
			// Signal that output job data has been updated
			stConfigOut.DataChange := stConfigOut.DataChange + 1;
	
		ELSE
			// Wrong configuration data type!
			stConfigOut.ConfigurationType := '';
			stConfigOut.DateTime := SYSTEMTIME_TO_DT(timestr:=fbGetTime.TIMESTR);
	
			// Signal that configuration data has been written		
			stConfigOut.ChangeStatus := stConfigIn.ChangeRequest;
			
			// Signal that output configuration data has been updated
			stConfigOut.DataChange := stConfigOut.DataChange + 1;
	
		END_IF
	END_IF
END_IF


// Upcoming Configuration
IF (stUpcomingConfigIn.ChangeRequest <> stUpcomingConfigOut.ChangeStatus) AND (stUpcomingConfigIn.ChangeRequest > 0) THEN
	sTempString := CONCAT('Upcoming ConfigChange request - Old request: ', TO_STRING(stUpcomingConfigOut.ChangeStatus));
	sTempString := CONCAT(sTempString, ', New request: ');
	sTempString := CONCAT(sTempString, TO_STRING(stUpcomingConfigIn.ChangeRequest));
	sTempString := CONCAT(sTempString, ' ConfigType: ');
	F_LogFile(CONCAT(sTempString, stUpcomingConfigIn.ConfigurationType)); 	

	// Change request from Line Controller
	IF (stAdditionalDataIn.MESHandShakes.DataChangeStatusUpcomingConfiguration = stUpcomingConfigOut.DataChange) THEN
		stUpcomingConfigOut.ChangeAcknowledge := stUpcomingConfigIn.ChangeRequest;
		stUpcomingConfigOut.DataChange := stUpcomingConfigOut.DataChange + 1;
	
		// Check Configuration Type
		IF (F_StringCompNoCase(stUpcomingConfigIn.ConfigurationType, 'OP11600')) THEN	
			// Update configuration data
			stUpcomingConfigOut.ConfigurationType := stUpcomingConfigIn.ConfigurationType;
			stConfigOut.DateTime := SYSTEMTIME_TO_DT(timestr:=fbGetTime.TIMESTR);
			stUpcomingConfigOut.OP11600 := stUpcomingConfigIn.OP11600;
	
			// Signal that configuration data has been written		
			stUpcomingConfigOut.ChangeStatus := stUpcomingConfigIn.ChangeRequest;
			
			// Signal that output configuration data has been updated
			stUpcomingConfigOut.DataChange := stUpcomingConfigOut.DataChange + 1;
			
		ELSE
			// Wrong configuration data type!
			stUpcomingConfigOut.ConfigurationType := '';
			stConfigOut.DateTime := SYSTEMTIME_TO_DT(timestr:=fbGetTime.TIMESTR);
	
			// Signal that configuration data has been written		
			stUpcomingConfigOut.ChangeStatus := stUpcomingConfigIn.ChangeRequest;
			
			// Signal that output configuration data has been updated
			stUpcomingConfigOut.DataChange := stUpcomingConfigOut.DataChange + 1;
	
		END_IF
	END_IF
END_IF
END_METHOD

METHOD M_DeviceDriver
VAR_INPUT
END_VAR
VAR

END_VAR

fbHS_Driver.P_bSimulationMode := stControlIn.General.SimulationMode;
fbHS_Driver.P_stCellCommandData := stHSDriverWrite;
fbHS_Driver();
stHSDriverRead := fbHS_Driver.P_stCellStatusData;

//Set device using idle setting
IF (eCurrentState = E_PMLState.ePMLState_Idle AND (aVehiclesStationFIFO[1].sCarrierID = '')) THEN
	stHSDriverWrite.rSetTemp := stControlIn.OP11600.IdleTemperature;
	stHSDriverWrite.rSetSteamReq := 0;
	stHSDriverWrite.rSetFanSpeed := stControlIn.OP11600.IdleFanSpeed;
END_IF

//Start timer until ModeState = Stop
IF eCurrentState = E_PMLState.ePMLState_Idle THEN
	tonIdleTimer.IN := ( (stReservation.nTicket = 0) AND (aVehiclesStationFIFO[1].sCarrierID = '') );

	IF tonIdleTimer.Q THEN
		bStopLocal := TRUE;
		
		F_Logfile('STAT1: Idle timer timed out, stop local');
	END_IF
ELSE
	tonIdleTimer.IN := FALSE;
END_IF

tonIdleTimer(IN:= , PT:= TO_TIME(stControlIn.General.StationIdleTime * 60000), Q=> , ET=> );
END_METHOD

METHOD PROTECTED M_ErrorWarning
VAR_INPUT
END_VAR
VAR
	bDataChange:BOOL;
END_VAR

bDataChange S= 
M_ErrorWarningObj(arErrorWaringData:= stErrorWarning.ErrorWarningData,
	bActive:= stHSDriverRead.stAlarms.TEMP_PROBE_FAULT, 
	iErrorWarningType:= 2, 
	diErrorWarningID:= E_AlarmCategory.OP11600 + 0, 
	sDeviceID:= 'OP11600',
	iSeverity:= 2, 
	iNativeID:= 0, 
	sNativeMessage:= 'Temperatur probe fault');
	
bDataChange S= 
M_ErrorWarningObj(arErrorWaringData:= stErrorWarning.ErrorWarningData,
	bActive:= stHSDriverRead.stAlarms.FAULT_INVERTER, 
	iErrorWarningType:= 2, 
	diErrorWarningID:= E_AlarmCategory.OP11600 + 1, 
	sDeviceID:= 'OP11600',
	iSeverity:= 2, 
	iNativeID:= 1, 
	sNativeMessage:= 'Fault inverter');

bDataChange S= 
M_ErrorWarningObj(arErrorWaringData:= stErrorWarning.ErrorWarningData,
	bActive:= stHSDriverRead.stAlarms.ENERGY_METER_COM_ERROR, 
	iErrorWarningType:= 1, 
	diErrorWarningID:= E_AlarmCategory.OP11600 + 6, 
	sDeviceID:= 'OP11600',
	iSeverity:= 1, 
	iNativeID:= 6, 
	sNativeMessage:= 'Energy meter comm. error');
	
bDataChange S= 
M_ErrorWarningObj(arErrorWaringData:= stErrorWarning.ErrorWarningData,
	bActive:= stHSDriverRead.eMachStatus = E_EMS_HS_Status.ALARM, 
	iErrorWarningType:= 2, 
	diErrorWarningID:= E_AlarmCategory.OP11600 + 16, 
	sDeviceID:= 'OP11600',
	iSeverity:= 2, 
	iNativeID:= 0, 
	sNativeMessage:= 'Device in Alarm');
	
bDataChange S= 
M_ErrorWarningObj(arErrorWaringData:= stErrorWarning.ErrorWarningData,
	bActive:= NOT stHSDriverRead.stStates.REMOTE_MODE, 
	iErrorWarningType:= 1, 
	diErrorWarningID:= E_AlarmCategory.OP11600 + 17, 
	sDeviceID:= 'OP11600',
	iSeverity:= 1, 
	iNativeID:= 0, 
	sNativeMessage:= 'Device in Local mode');
	
bDataChange S= 
M_ErrorWarningObj(arErrorWaringData:= stErrorWarning.ErrorWarningData,
	bActive:= stHSDriverRead.stStates.ALARM_IN_PROGRESS, 
	iErrorWarningType:= 1, 
	diErrorWarningID:= E_AlarmCategory.OP11600 + 18, 
	sDeviceID:= 'OP11600',
	iSeverity:= 1, 
	iNativeID:= 0, 
	sNativeMessage:= 'Deivce Alarm in progress');


stErrorWarning.DataChange := stErrorWarning.DataChange + TO_UINT(bDataChange);
bDataChange := FALSE;
END_METHOD

/// Static state "Execute"
/// Trigged by "StageCompleted" when in "Starting" state
/// Trigged by "StageCompleted" when in "Unholding" state
/// Trigged by "StageCompleted" when in "Unsuspending" state
/// Requires "Hold" command to go to "Holding" state 
/// Requires "Suspend" command to go to "Suspending" state 
/// Requires "StageCompleted" to go to "Completing" state 
{attribute 'object_name' := 'M_Execute'}
METHOD M_Execute
VAR
	i		: UINT;
	sTempString : STRING(200);
	fTMachineMid : REAL;
	fSMachineMid : REAL;
	fAMachineMid : REAL;
END_VAR
// Sequence
//Run current cycle duration timer
IF diStateTImer < 1000000 THEN
	diStateTimer := diStateTimer + g_iPLCScan_MS;
END_IF

//New Vehicle in device fifo location
FOR i := 1 TO 9 DO
	IF (aVehiclesStationFIFO[i+1].sCarrierID = '') THEN
		EXIT;
	END_IF
END_FOR
iVehicleInFIFO := i;

CASE eSeq OF
	E_HSStationINSeq.Idle:
		diStateTimer := 0;
		
		IF bVehicleReadyAtInput OR bSkipVehicle THEN
			eSeq := E_HSStationINSeq.NewJob;
			
			F_Logfile('STAT1: Vehicle ready');
		END_IF
	
	E_HSStationINSeq.NewJob:		
		//Check for other vehicles in device				
		IF iVehicleInFIFO = 1 THEN //New vehicle is only vehicle in FIFO
			IF bSkipVehicle THEN
				eSeq := E_HSStationINSeq.ReceiveNextVehicle;
				F_LogFile('STAT1: Skip job - No other carriers in device');
			ELSE
				eSeq := E_HSStationINSeq.SetSettingsOnDevice;//No items in FIFO
				F_LogFile('STAT1: new job - No other carriers in device');
			END_IF
			
		ELSIF iVehicleInFIFO > 1 THEN //More vehicles in FIFO
			eSeq := E_HSStationINSeq.CheckVehiclesVelocity;				
			F_LogFile(CONCAT('STAT1: new job - Carrier ID: ', TO_STRING(aVehiclesStationFIFO[iVehicleInFIFO].sCarrierID)));
		END_IF

	E_HSStationINSeq.CheckVehiclesVelocity:
		IF iVehicleInFIFO > 1 AND NOT bSkipVehicle THEN
			IF ( (aVehiclesStationFIFO[iVehicleInFIFO-1].fCalculatedTIA > fTimeCal) ) THEN
				IF bStateChange_OS THEN
					sTempString := (CONCAT('STAT1: Vehicle with Carrier ID: ', TO_STRING(aVehiclesStationFIFO[iVehicleInFIFO].sCarrierID)));
					sTempString := CONCAT(sTempString, ', Calc. TIA: ');
					sTempString := CONCAT(sTempString, TO_STRING(fTimeCal));
					sTempString := CONCAT(sTempString, ', Faster than: ');
					sTempString := CONCAT(sTempString, TO_STRING(aVehiclesStationFIFO[i].sCarrierID));
					sTempString := CONCAT(sTempString, ', With TIA: ');
					F_LogFile(CONCAT(sTempString, TO_STRING(aVehiclesStationFIFO[i].fCalculatedTIA)));
				END_IF
			ELSE
				eSeq := E_HSStationINSeq.CheckVehiclesSettings;
						
				sTempString := CONCAT('STAT1: Vehicle with Carrier ID: ', TO_STRING(sCarrierID));
				sTempString := CONCAT(sTempString, ', Calc. TIA: ');
				sTempString := CONCAT(sTempString, TO_STRING(fTimeCal));
				F_Logfile(CONCAT(sTempString, ', Velocity OK to enter'));
			END_IF
		ELSIF iVehicleInFIFO <= 1 THEN
			eSeq := E_HSStationINSeq.SetSettingsOnDevice;//No items in FIFO
			F_LogFile('STAT1: No other carriers in device');
		ELSIF bSkipVehicle THEN // Skip vehicle - interpolate velocity with previous vehicle
			IF (aVehiclesStationFIFO[iVehicleInFIFO-1].fCalculatedTIA > 0) THEN
				aVehiclesStationFIFO[iVehicleInFIFO].fVelocity := LIMIT(0.001,(sDistanceInDevice / aVehiclesStationFIFO[iVehicleInFIFO-1].fCalculatedTIA), 1);
			ELSE
				aVehiclesStationFIFO[iVehicleInFIFO].fVelocity := 1;
			END_IF
			fVelocityCal := aVehiclesStationFIFO[iVehicleInFIFO].fVelocity; //set velocity
			eSeq := E_HSStationINSeq.ReceiveNextVehicle;
			F_LogFile(CONCAT('STAT1: Skip, vehicle vel. set to: ', REAL_TO_STRING(aVehiclesStationFIFO[iVehicleInFIFO].fVelocity)));
		END_IF
	
	E_HSStationINSeq.CheckVehiclesSettings:
		fTMachineMid:= stJobDataOut.OP11600.TemperatureMax + stJobDataOut.OP11600.TemperatureMin;
		IF fTMachineMid > 0 THEN
			fTMachineMid := fTMachineMid/2;
		END_IF
		
		fSMachineMid:= stJobDataOut.OP11600.SteamMax + stJobDataOut.OP11600.SteamMin;
		IF fSMachineMid > 0 THEN
			fSMachineMid := fSMachineMid/2;
		END_IF
		
		fAMachineMid:= stJobDataOut.OP11600.AirMax + stJobDataOut.OP11600.AirMin;
		IF fAMachineMid > 0 THEN
			fAMachineMid := fAMachineMid/2;
		END_IF
		FOR i := 1 TO 10 DO
			IF (aVehiclesStationFIFO[i].sCarrierID <> '') THEN
				
				IF (fTMachineMid) > aVehiclesStationFIFO[i].JobData.TemperatureMax OR
					(fTMachineMid) < aVehiclesStationFIFO[i].JobData.TemperatureMin OR
					(fSMachineMid) > aVehiclesStationFIFO[i].JobData.SteamMax OR
					(fSMachineMid) < aVehiclesStationFIFO[i].JobData.SteamMin OR
					(fAMachineMid) > aVehiclesStationFIFO[i].JobData.AirMax OR
					(fAMachineMid) < aVehiclesStationFIFO[i].JobData.AirMin THEN
					
						IF bStateChange_OS THEN
							sTempString := (CONCAT('STAT1: Vehicle with Carrier ID: ', TO_STRING(aVehiclesStationFIFO[iVehicleInFIFO].sCarrierID)));
							F_LogFIle(CONCAT(sTempString, ', Check settings failed to enter'));
						END_IF
						
						EXIT; //End loop - at least 1 vehicle cannot accomodate settings
				END_IF
			ELSE
				sTempString := (CONCAT('STAT1: Vehicle with Carrier ID: ', TO_STRING(aVehiclesStationFIFO[iVehicleInFIFO].sCarrierID)));
				F_LogFIle(CONCAT(sTempString, ', Check settings OK to enter'));
				
				eSeq := E_HSStationINSeq.SetSettingsOnDevice;
				EXIT; //End reached
			END_IF
		END_FOR

	E_HSStationINSeq.SetSettingsOnDevice: (* Temperature limits 80-180C, Steam limits 0-10, Air flow limits 1500-3000*) 

		stHSDriverWrite.rSetTemp := LIMIT(80, fTemperatureCal, 180);
		stHSDriverWrite.rSetSteamReq := TO_DINT(LIMIT(0, fSteamCal, 10));
		stHSDriverWrite.rSetFanSpeed := LIMIT(1500, fAirCal, 3000);
		stHSDriverWrite.stCommands.REMOTE_START := TRUE;
		stHSDriverWrite.stCommands.REMOTE_STOP := FALSE;
		eSeq := E_HSStationINSeq.WaitForDeviceReady;
		
		sTempString := (CONCAT('STAT1: Vehicle with Carrier ID: ', TO_STRING(aVehiclesStationFIFO[iVehicleInFIFO].sCarrierID)));
		F_LogFIle(CONCAT(sTempString, ', Set settings on Barrera'));
		
	E_HSStationINSeq.WaitForDeviceReady:	
		//Wait for temperature reached
		IF (bTestActive OR (stHSDriverRead.rActTempVal >= stHSDriverWrite.rSetTemp - 10 AND stHSDriverRead.rActTempVal <= stHSDriverWrite.rSetTemp + 10) ) THEN
			eSeq := E_HSStationINSeq.ReceiveNextVehicle;
			
			sTempString := (CONCAT('STAT1: Vehicle with Carrier ID: ', TO_STRING(aVehiclesStationFIFO[iVehicleInFIFO].sCarrierID)));
			F_LogFIle(CONCAT(sTempString, ', Temp and steam setpoint reacehd'));
		END_IF
	
	E_HSStationINSeq.ReceiveNextVehicle:
		//Let cell release next vehicle with defined velocity
		eSeq := E_HSStationINSeq.Done;
		
			F_LogFile('STAT1: ready next vehicle');
		
	E_HSStationINSeq.Done:
				 
		 // Set job state to LC
		IF (stJobDataOut.JobState <> 3) AND NOT bSkipVehicle THEN
			stJobDataOut.JobState := 3; //(0: Undefined, 1: Idle, 2: Executing, 3: Completed)
			stJobDataOut.DataChange := stJobDataOut.DataChange + 1;
			IF (NOT bSkipVehicle) THEN
				M_OEEProductProcessed(TRUE);
			END_IF
		END_IF
	
		// Completed operation
		IF (iNextJobStation = 1 OR iNextJobStation = 2 OR bSkipVehicle)  THEN
			// Signal to Track system that operation(s) are completed - vehicle is already gone on this machine
			IF iNextJobStation = 1 OR iNextJobStation = 2 THEN
				F_LogFile(CONCAT('Cell4 - DONE(iNextJobStation = 1 or 2), Step: ', TO_STRING(eSeq)));
			ELSIF bSkipVehicle THEN
				F_LogFile(CONCAT('Cell4 - DONE(Skipped), Step: ', TO_STRING(eSeq)));
			END_IF
			
			iNextJobStation := 0;
			
			
			eSeq := E_HSStationINSeq.Idle;
			M_StateComplete();
		END_IF
END_CASE


bStateChange_OS := eSeq <> eSeq_Old;
eSeq_Old := eSeq;
END_METHOD

METHOD M_ExternalStart
VAR_INPUT
END_VAR
bStartLocal := TRUE;
END_METHOD

/// Static state "Held"
/// Trigged by "StateCompleted" when in "Holding" state
/// Requires "Unhold" command to go to "Unholding" state 
{attribute 'object_name' := 'M_Held'}
METHOD M_Held
END_METHOD

/// Dynamic state "Holding"
/// Trigged by "Hold" command when in "Execute" state
/// Requires "StateCompleted" to go to "Held" state 
{attribute 'object_name' := 'M_Holding'}
METHOD M_Holding

 M_StateComplete();
END_METHOD

/// Static state "Idle"
/// Trigged by "StateCompleted" when in "Resetting" state
/// Requires "Start" command to go to "Starting" state 
{attribute 'object_name' := 'M_Idle'}
METHOD M_Idle

VAR

END_VAR
// Set job state to LC
IF (stJobDataOut.JobState <> 1) THEN
	stJobDataOut.JobState := 1;//(0: Undefined, 1: Idle, 2: Executing, 3: Completed)
	stJobDataOut.DataChange := stJobDataOut.DataChange + 1;
END_IF

//Handle nextjobstation request
//IF (bVehicleReadyAtInput) THEN
	IF iNextJobStation <> iNextJobStationOld THEN
		f_LogFile(CONCAT('NextJobStation request: ', TO_STRING(iNextJobStation)));
		
		M_SetVelocity();
		
		//Skip Carrier
		IF iNextJobStation = 1 THEN
			bSkipVehicle := TRUE;
			bStartLocal := TRUE;
			iNextJobStation := 0;
		ELSIF iNextJobStation = 2 THEN
			;//Wait for start from LC
		END_IF
	END_IF
//END_IF

iNextJobStationOld := iNextJobStation;
END_METHOD

METHOD PROTECTED M_Init : BOOL;
VAR_INPUT
END_VAR
IF (NOT bInitDone) THEN
	// Call method in base FB
	SUPER^.M_Init();
		
	//Set ip to Barrera Heat and steam
	fbHS_Driver.P_ModbusIPBarrera := '10.38.190.221';

// Specify operational data
	stOperationalDataOut.OP11600.DeviceData[1] := F_NewDeviceDataX(	'HS',				'Heat & Steam',
																	11600+1,			'Temperature',		E_Units._degC	);
	stOperationalDataOut.OP11600.DeviceData[2] := F_NewDeviceDataX(	'HS',				'Heat & Steam',
																	11600+2,			'Steam',			E_Units.None	);
	stOperationalDataOut.OP11600.DeviceData[3] := F_NewDeviceDataX(	'HS',				'Heat & Steam',
																	11600+3,			'Fan speed',		E_Units._RPM	);
	stOperationalDataOut.OP11600.DeviceData[4] := F_NewDeviceDataX(	'HS',				'Heat & Steam',
																	11600+4,			'Power',			E_Units._KW	);
	stOperationalDataOut.OP11600.DeviceData[5] := F_NewDeviceDataX(	'HS',				'Heat & Steam',
																	11600+5,			'Energy',			E_Units._KWh	);
	stOperationalDataOut.OP11600.DeviceData[6] := F_NewDeviceDataX(	'HS',				'Heat & Steam',
																	11600+6,			'Running hours',	E_Units._hour	);
	stOperationalDataOut.OP11600.DeviceData[7] := F_NewDeviceDataX(	'HS',				'Heat & Steam',
																	11600+7,			'Running minutes',	E_Units._min	);

	bInitDone := TRUE;
END_IF
END_METHOD

METHOD M_JobDataHandling
VAR_INPUT
END_VAR
VAR
	sTempString : STRING(200);
END_VAR
// Job Data to device
IF (stJobDataIn.ChangeRequest <> stJobDataOut.ChangeStatus) AND (stJobDataIn.ChangeRequest > 0) THEN
	sTempString := CONCAT('NewJobdata request - Old request: ', TO_STRING(stJobDataOut.ChangeStatus));
	sTempString := CONCAT(sTempString, ', New request: ');
	sTempString := CONCAT(sTempString, TO_STRING(stJobDataIn.ChangeRequest));
	sTempString := CONCAT(sTempString, ' JobDataType: ');
	sTempString := CONCAT(sTempString, stJobDataIn.JobDataType); 	

	// Change request from Line Controller
	// Check if LC allows data output change
	IF (stAdditionalDataIn.MESHandShakes.DataChangeStatusJobData = stJobDataOut.DataChange) THEN
// NOTE: Changed to match new LC software!!! - Hack!				
//		stJobDataOut.ChangeAcknowledge := stJobDataIn.ChangeRequest;
//		stJobDataOut.DataChange := stJobDataOut.DataChange + 1;
	
		// Next job station (operator decision)
		iNextJobStation := stJobDataIn.NextJobStation;
	
		// Check Job Type
		IF (F_StringCompNoCase(stJobDataIn.JobDataType, 'OP11600')) THEN	
	
			// Update output job data
			stJobDataOut.OP11600 := stJobDataIn.OP11600;
			stJobDataOut.JobDataType := stJobDataIn.JobDataType;
	
			// Signal that job data has been written		
// NOTE: Changed to match new LC software!!! - Hack!				
			stJobDataOut.ChangeAcknowledge := stJobDataIn.ChangeRequest;
			stJobDataOut.ChangeStatus := stJobDataIn.ChangeRequest;
			
			// Set job state to Idle
			stJobDataOut.JobState := 1;
			
			// Signal that output job data has been updated
			stJobDataOut.DataChange := stJobDataOut.DataChange + 1;
	
		ELSE
	
			// Update output job data
			stJobDataOut.JobDataType := '';
	
			// Signal that job data has been written		
// NOTE: Changed to match new LC software!!! - Hack!				
			stJobDataOut.ChangeAcknowledge := stJobDataIn.ChangeRequest;
			stJobDataOut.ChangeStatus := stJobDataIn.ChangeRequest;
			
			// Signal that output job data has been updated
			stJobDataOut.DataChange := stJobDataOut.DataChange + 1;
	
		END_IF
	END_IF
	
	sTempString := CONCAT(sTempString, ', TTarget: ');
	sTempString := CONCAT(sTempString, TO_STRING(stJobDataIn.OP11600.TemperatureTarget));
	sTempString := CONCAT(sTempString, ', TMin: ');
	sTempString := CONCAT(sTempString, TO_STRING(stJobDataIn.OP11600.TemperatureMin));
	sTempString := CONCAT(sTempString, ', TMax: ');
	sTempString := CONCAT(sTempString, TO_STRING(stJobDataIn.OP11600.TemperatureMax));
	sTempString := CONCAT(sTempString, ', SMin: ');
	sTempString := CONCAT(sTempString, TO_STRING(stJobDataIn.OP11600.SteamMin));
	sTempString := CONCAT(sTempString, ', SMax: ');
	sTempString := CONCAT(sTempString, TO_STRING(stJobDataIn.OP11600.SteamMax));
	sTempString := CONCAT(sTempString, ', AMin: ');
	sTempString := CONCAT(sTempString, TO_STRING(stJobDataIn.OP11600.AirMin));
	sTempString := CONCAT(sTempString, ', AMax: ');
	F_LogFile(CONCAT(sTempString, TO_STRING(stJobDataIn.OP11600.AirMax)));
END_IF
END_METHOD

METHOD PROTECTED M_OperationalDataHandling
VAR
END_VAR
// Check if LC allows data output change
IF (stAdditionalDataIn.MESHandShakes.DataChangeStatusOperationalData = stOperationalDataOut.DataChange) THEN
	// Heat and Steam
	stOperationalDataOut.OP11600.DeviceData[1].Value := stHSDriverRead.rActTempVal;
	stOperationalDataOut.OP11600.DeviceData[2].Value := stHSDriverRead.rActSteamReq;
	stOperationalDataOut.OP11600.DeviceData[3].Value := (BIT_TO_REAL(stHSDriverRead.stStates.MACHINE_READY_TO_WORK) * stHSDriverRead.rActFanReq);
	stOperationalDataOut.OP11600.DeviceData[4].Value := stHSDriverRead.rInstPower;
	stOperationalDataOut.OP11600.DeviceData[5].Value := stHSDriverRead.rEnergyCons;
	stOperationalDataOut.OP11600.DeviceData[6].Value := stHSDriverRead.iRunningHrs;
	stOperationalDataOut.OP11600.DeviceData[7].Value := stHSDriverRead.iRunningMins;
	
END_IF
END_METHOD

/// Dynamic state "Resetting"
/// Trigged by "Reset" command when in "Stopped" state
/// Requires "StateCompleted" to go to "Idle" state 
{attribute 'object_name' := 'M_Resetting'}
METHOD M_Resetting
M_StateComplete();

//Update jobdata
IF NOT bSkipVehicle THEN
	stJobDataOut.DataChange := stJobDataOut.DataChange +1;
	stJobDataOut.JobState	:= 1; //(0: Undefined, 1: Idle, 2: Executing, 3: Completed)
END_IF
bSkipVehicle := FALSE;

// Reset next job station value before entering Idle state
iNextJobStation := 0;
iNextJobStationOld := 0;

//Set idle settings - station empty
IF (aVehiclesStationFIFO[1].sCarrierID = '') THEN
	stHSDriverWrite.rSetTemp := stControlIn.OP11600.IdleTemperature;
	stHSDriverWrite.rSetSteamReq := 0;
	stHSDriverWrite.rSetFanSpeed := stControlIn.OP11600.IdleFanSpeed;
	stHSDriverWrite.stCommands.REMOTE_START := TRUE;
	stHSDriverWrite.stCommands.REMOTE_STOP := FALSE;
END_IF

bResetLocal := FALSE;
END_METHOD

METHOD PRIVATE M_SetVelocity : REAL;
VAR_INPUT
END_VAR
VAR
	sTempString	:STRING(200);
END_VAR
//Calculate velocity
IF stJobDataIn.NextJobStation = 2 THEN

	// Calculate velocity and machine temperature
	F_CalcValuesHeatSteam(	rTempFinal:= stJobDataIn.OP11600.TemperatureTarget, 
							rTempInitial:= stAdditionalDataIn.OP11600.TempInitial, 
							rCT:= stJobDataIn.OP11600.Profile[1], 
							rCS:= stJobDataIn.OP11600.Profile[2], 
							rCA:= stJobDataIn.OP11600.Profile[3], 
							rMachineLength:= sDistanceInDevice, 
							rTimeMin:= stJobDataIn.OP11600.TimeMin, 
							rTimeMax:= stJobDataIn.OP11600.TimeMax, 
							rTempMin:= stJobDataIn.OP11600.TemperatureMin, 
							rTempMax:= stJobDataIn.OP11600.TemperatureMax, 
							rSteamMin:= stJobDataIn.OP11600.SteamMin, 
							rSteamMax:= stJobDataIn.OP11600.SteamMax, 
							rAirMin:= stJobDataIn.OP11600.AirMin, 
							rAirMax:= stJobDataIn.OP11600.AirMax, 
							rVelocity=> fVelocityCal, 
							rTempMachine=> fTemperatureCal, 
							rSteamMachine=> fSteamCal,
							rAirMachine=> fAirCal,
							rTimeMachine=> fTimeCal 	);

ELSE
	fVelocityCal := 1;
	sTempString := CONCAT('STAT1: SetVelocity - fixed velocity due to skip: ', TO_STRING(fVelocityCal));
	F_Logfile(sTempString);

END_IF		

M_SetVelocity := fVelocityCal;
END_METHOD

METHOD PRIVATE M_SetVelocity_OLD : REAL;
VAR_INPUT
END_VAR
VAR
	sTempString	:STRING(200);
	fTMachineMid : REAL;
	fSMachineMid : REAL;
	fAMachineMid : REAL;
	sTempVelocity:STRING;
END_VAR
//Calculate velocity
IF stJobDataIn.NextJobStation = 2 THEN (* Temperature limits 80-180C, Steam limits 0-10, Air flow limits 1500-3000*)

	IF ( (stJobDataIn.OP11600.Profile[1] = 0.0) AND
		 (stJobDataIn.OP11600.Profile[2] = 0.0) AND
		 (stJobDataIn.OP11600.Profile[3] = 0.0) ) THEN
		// Use min time in machine and max device allowed settings from job data
		F_Logfile('SetVelocity - COeffs ZERO, use MAX settings and MIN time');
		
		//Calculate time needed in machine
		IF (stJobDataIn.OP11600.TimeMin > 0) THEN
			fCalcTimeInDevice := stJobDataIn.OP11600.TimeMin;
		ELSIF (stJobDataIn.OP11600.TimeMax > 0) THEN
			fCalcTimeInDevice := stJobDataIn.OP11600.TimeMax;
		ELSE
			// Default valie 2 minutes
			fCalcTimeInDevice := 120;
		END_IF
		
		fCalcTimeInDeviceLimits := fCalcTimeInDevice;

	ELSE
		F_Logfile('SetVelocity - COeffs OK, Calculate velocity');

		fTMachineMid:= stJobDataIn.OP11600.TemperatureMax + stJobDataIn.OP11600.TemperatureMin;
		IF fTMachineMid > 0 THEN
			fTMachineMid := fTMachineMid/2;
		END_IF
		
		fSMachineMid:= stJobDataIn.OP11600.SteamMax + stJobDataIn.OP11600.SteamMin;
		IF fSMachineMid > 0 THEN
			fSMachineMid := fSMachineMid/2;
		END_IF
		
		fAMachineMid:= stJobDataIn.OP11600.AirMax + stJobDataIn.OP11600.AirMin;
		IF fAMachineMid > 0 THEN
			fAMachineMid := fAMachineMid/2;
		END_IF
	
		M_SetVelocity := M_CalculatedVelocity(
								fTFinal:= stJobDataIn.OP11600.TemperatureTarget, 
								fTInital:= 20, //where to get initial temperature?? 
								fTMachine:= LIMIT(80, fTMachineMid, 180), 
								fSMachine:= LIMIT(0, fSMachineMid, 10), 
								fAMachine:= LIMIT(1500, fAMachineMid, 3000), 
								fcT:= stJobDataIn.OP11600.Profile[1], 
								fcS:= stJobDataIn.OP11600.Profile[2], 
								fcA:= stJobDataIn.OP11600.Profile[3], 
								fTravelLength:= sDistanceInDevice);
	
		sTempString := CONCAT('SetVelocity - Vel. Calc raw: ', TO_STRING(M_SetVelocity));
						
		//Velocity limit on MagneMotion
		M_SetVelocity := LIMIT(0.001, M_SetVelocity, 2); 
		
		//Calculate time needed in machine
		fCalcTimeInDevice := sDistanceInDevice / M_SetVelocity;
		
		//Check with limits
		fCalcTimeInDeviceLimits := LIMIT(stJobDataIn.OP11600.TimeMin, fCalcTimeInDevice, stJobDataIn.OP11600.TimeMax);

	END_IF
	
	//Calculated velocity with time limits
	fVelocityCalLimits := sDistanceInDevice / fCalcTimeInDeviceLimits;
	
	M_SetVelocity := LIMIT(0.001, fVelocityCalLimits, 2);
	
	sTempString := CONCAT(sTempString, ', Velocity Calc: ');
	sTempString := CONCAT(sTempString, TO_STRING(M_SetVelocity));
	sTempString := CONCAT(sTempString, ', Time in machine: ');
	sTempString := CONCAT(sTempString, TO_STRING(fCalcTimeInDeviceLimits));
	F_Logfile(sTempString);
ELSE
	M_SetVelocity := 1;
	sTempString := CONCAT('SetVelocity - fixed velocity due to skip: ', TO_STRING(M_SetVelocity));
	F_Logfile(sTempString);
END_IF
END_METHOD

/// Dynamic state "Starting"
/// Trigged by "Start" command when in "Idle" state
/// Requires "StateCompleted" to go to "Execute" state 
{attribute 'object_name' := 'M_Starting'}
METHOD M_Starting
// Starting production mode

//Update jobdata
IF stJobDataOut.JobState <> 2 AND NOT bSkipVehicle THEN
	stJobDataOut.DataChange := stJobDataOut.DataChange +1;
	stJobDataOut.JobState := 2; //(0: Undefined, 1: Idle, 2: Executing, 3: Completed)
END_IF

// Start execute sequence
iNextJobStation := 0;
bStartLocal := FALSE;
eCommand := E_PML_Command.Undefined;
eSeq := E_HSStationINSeq.Idle;

//Wait for Carrier ID on station are different than last carrierID and CarrierID appears in FIFO
IF (stVehicleDataStaion.stVehicle.sCarrierID <> '') (*AND stVehicleDataStaion.stVehicle.sCarrierID <> sCarrierID*) (*AND NOT bSkipVehicle*) THEN
	FOR i := 1 TO 10 DO
		IF stVehicleDataStaion.stVehicle.sCarrierID = aVehiclesStationFIFO[i].sCarrierID THEN
			sCarrierID := stVehicleDataStaion.stVehicle.sCarrierID; //Update for comparison
			M_StateComplete();
			EXIT;
		END_IF
	END_FOR
//ELSIF bSkipVehicle THEN
//	M_StateComplete();
END_IF
END_METHOD

/// Static state "Stopped"
/// Trigged by "StateCompleted" when in "Stopping" state
/// Requires "Reset" command to go to "Resetting" state 
{attribute 'object_name' := 'M_Stopped'}
METHOD M_Stopped
IF stReservation.nTicket <> 0 THEN
	bResetLocal := TRUE;
	
	F_Logfile('STAT1: Reservation list updated, reset local');
END_IF
END_METHOD

/// Dynamic state "Stopping"
/// Trigged by "Stop" command
/// Requires "StateCompleted" to go to "Stopped" state 
{attribute 'object_name' := 'M_Stopping'}
METHOD M_Stopping

stHSDriverWrite.rSetFanSpeed := 0;
stHSDriverWrite.rSetTemp := 0;
stHSDriverWrite.stCommands.REMOTE_STOP := TRUE;
stHSDriverWrite.stCommands.REMOTE_START := FALSE;
bStopLocal := FALSE;

 M_StateComplete();
END_METHOD

/// Static state "Suspended"
/// Trigged by "StateCompleted" when in "Suspending" state
/// Requires "Unsuspend" command to go to "Unsuspending" state 
{attribute 'object_name' := 'M_Suspended'}
METHOD M_Suspended
END_METHOD

/// Dynamic state "Suspending"
/// Trigged by "Suspend" command when in "Execute" state
/// Requires "StateCompleted" to go to "Suspended" state 
{attribute 'object_name' := 'M_Suspending'}
METHOD M_Suspending

 M_StateComplete();
END_METHOD

/// Dynamic state "Unholding"
/// Trigged by "Unhold" command when in "Held" state
/// Requires "StateCompleted" to go to "Execute" state 
{attribute 'object_name' := 'M_Unholding'}
METHOD M_Unholding

 M_StateComplete();
END_METHOD

/// Dynamic state "Unsuspending"
/// Trigged by "Unsuspend" command when in "Suspended" state
/// Requires "StateCompleted" to go to "Execute" state 
{attribute 'object_name' := 'M_Unsuspending'}
METHOD M_Unsuspending

 M_StateComplete();
END_METHOD

PROPERTY P_bSkipVehicle : BOOL
GET
P_bSkipVehicle := bSkipVehicle;
END_GET
SET
bSkipVehicle := P_bSkipVehicle;
END_SET
END_PROPERTY

END_FUNCTION_BLOCK

// ---- ECC/Basic/Station/FB_Station_Basic.TcPOU
/// Generic FB for cells/stations
/// Contains the PackML state machine and PackTags data
FUNCTION_BLOCK FB_Station_Basic IMPLEMENTS ITF_UnitState 
VAR_INPUT
	nCellStateCmd			: E_PML_Command;			// Cell PML state command
	bVehicleReadyAtInput	: BOOL;						// Set to TRUE when a vehicle is ready at the station input location
	bVehicleReadyAtOutput	: BOOL;						// Set to TRUE when a vehicle is ready at the station output location
END_VAR
VAR_OUTPUT
	bUndefinedDone			: BOOL;						// When the SPS is started, the first state is Undefiend. bUndefinedDone is TRUE, when the method Undefined has succesful finished
	bInvalidModeCommandOut	: BOOL;
	bChangeIntoProduction	: BOOL;
	bStationCommError		: BOOL := FALSE;			// Error communication with station PLC/HW
	UnitModeChangeInProcess	: BOOL;
	bReadyForVehicleInput	: BOOL;						// TRUE when station is ready for a vehicle/last at input location
	bCompletedInput			: BOOL;						// TRUE when part operation has finished (ready to deliver to vehicle on input)
	bReadyForVehicleOutput	: BOOL;						// TRUE when station is ready for a vehicle/last at output location
	bCompletedOutput		: BOOL;						// TRUE when part operation has finished (ready to deliver to vehicle on input)
END_VAR
VAR_IN_OUT
	stModeStateIn			: ST_InputModeState;
	stModeStateOut			: ST_OutputModeState;	
	stOEE					: ST_OutputOEE;
	stErrorWarning			: ST_OutputErrorWarning;
END_VAR
VAR
// Mode and State requests
	// Input:
	eMode					: E_PMLProtectedUnitMode := E_PMLProtectedUnitMode.ePMLProtUnitMode_Production;
	eCommand				: E_PMLCommand := E_PMLCommand.ePMLCommand_Undefined;
	bModeChangeRequest		: BOOL;
	// Output:
	eRequestedMode			: E_PMLProtectedUnitMode;
	eCurrentMode			: E_PMLProtectedUnitMode;
	eRequestedState			: E_PMLState;
	eCurrentState			: E_PMLState;	

// PackML
	fbUnitModeManager		: PML_UnitModeManager;		// The PML_UnitModeManager manage the Modechanges
	UnitModeChangeRequest	: BOOL;						// Set to TRUE to perform a mode change
	fbStateMachine 			: PML_StateMachine;			// The PML_StateMachine mangae the Statechanges
	nStateModeChange		: INT	:= 0;				// Variable to handle the modechange
	nLastState				: E_PMLState;				// Variable to store last state
	bProductionLocal		: BOOL := FALSE;			// Local Production mode button/command. Must be updated in inherited FB's
	bManualLocal			: BOOL := FALSE;			// Local Manual mode button/command. Must be updated in inherited FB's
	bMaintenanceLocal		: BOOL := FALSE;			// Local Maintenance mode button/command. Must be updated in inherited FB's
	bEStopOK				: BOOL := TRUE;				// TRUE when emergency stop is OK. Must be updated in inherited FB's
														// Will result in Abort state in PackML!
	bAbortLocal				: BOOL := FALSE;			// Local abort button/command. Must be updated in inherited FB's
	bStartLocal				: BOOL := FALSE;			// Local start button/command. Must be updated in inherited FB's
	bStopLocal				: BOOL := FALSE;			// Local stop button/command. Must be updated in inherited FB's
	bResetLocal				: BOOL := FALSE;			// Local reset button/command. Must be updated in inherited FB's
	bClearLocal				: BOOL := FALSE;			// Local clear button/command. Must be updated in inherited FB's
	bHoldLocal				: BOOL := FALSE;			// Local hold button/command. Must be updated in inherited FB's
	bUnholdLocal			: BOOL := FALSE;			// Local unhold button/command. Must be updated in inherited FB's
	bSuspendLocal			: BOOL := FALSE;			// Local suspend button/command. Must be updated in inherited FB's
	bUnsuspendLocal			: BOOL := FALSE;			// Local unsuspend button/command. Must be updated in inherited FB's

// Misc
	fbGetTime				: NT_GetTime;
	bInitDone				: BOOL;

END_VAR
VAR PERSISTENT
	iGoodProduct			: UDINT;					// For keeping values during power-off
	iProcessedProduct		: UDINT;					// Values are copied to stOEE in M_Init
	iRejectedProduct		: UDINT;					// 
END_VAR


// Init
M_Init();

// Get system time
fbGetTime(	NETID:= '',	// Local PLC 
			START:= NOT fbGetTime.START AND NOT fbGetTime.BUSY, 
			TMOUT:= T#5S	);

// Follow cellbridge states
CASE nCellStateCmd OF
	E_PML_Command.Reset,
	E_PML_Command.Hold,
	E_PML_Command.Unhold,
	E_PML_Command.Suspend,
	E_PML_Command.Unsuspend,
	E_PML_Command.Abort,
	E_PML_Command.Clear:
		// Station must follow cellbridge commands
		eCommand := nCellStateCmd;

	E_PML_Command.Start,
	E_PML_Command.Stop,
	E_PML_Command.Complete:
		;
END_CASE

// Mode state handshake handling
IF ((stModeStateIn.ChangeRequest <> stModeStateOut.ChangeStatus) AND (stModeStateIn.ChangeRequest > 0)) THEN
	// Mode change
	IF ( (stModeStateIn.Mode > 0) AND (stModeStateIn.Mode <= 6) ) THEN
		// Set acknowledge
		IF (stModeStateOut.ChangeAcknowledge <> stModeStateIn.ChangeRequest) THEN
			stModeStateOut.ChangeAcknowledge := stModeStateIn.ChangeRequest;
			stModeStateOut.ModeStateResponse := 0;
			stModeStateOut.DataChange := stModeStateOut.DataChange + 1;
		END_IF
		// Set new mode
		eMode := stModeStateIn.Mode;
		stModeStateOut.RequestedMode := DINT_TO_UINT(eMode);
		// Wait done
		IF (stModeStateIn.Mode = eCurrentMode) THEN
			// Set change status
			stModeStateOut.ChangeStatus := stModeStateIn.ChangeRequest;
			stModeStateOut.ModeStateResponse := 3;
			stModeStateOut.DataChange := stModeStateOut.DataChange + 1;
			stModeStateIn.Mode := E_PML_Mode.Undefined;
		END_IF
	END_IF

	// State change
	IF ( (stModeStateIn.State > 0) AND (stModeStateIn.State <= 10) ) THEN
		// Set acknowledge
		IF (stModeStateOut.ChangeAcknowledge <> stModeStateIn.ChangeRequest) THEN
			stModeStateOut.ChangeAcknowledge := stModeStateIn.ChangeRequest;
			stModeStateOut.ModeStateResponse := 0;
			stModeStateOut.DataChange := stModeStateOut.DataChange + 1;
		END_IF

		// Check job data when START command
		IF ( (stModeStateIn.State = E_PML_Command.Start) AND (stModeStateIn.State <> eCommand)) THEN
			IF (M_CheckJobData()) THEN
				// Job data OK! Set new state command
				F_LogLine('STAT: Check Jobdata OK', stModeStateIn.State);
				eCommand := stModeStateIn.State;
			ELSE
				// Job data NOT OK! Set change status to not possible to handle!
				F_LogLine('STAT: Check Jobdata failed', stModeStateIn.State);
				stModeStateOut.ChangeStatus := stModeStateIn.ChangeRequest;
				stModeStateOut.ModeStateResponse := 1;	// Could not handle START request!
				stModeStateOut.DataChange := stModeStateOut.DataChange + 1;
				stModeStateIn.State := E_PML_Command.Undefined;
				eCommand := E_PML_Command.Undefined;
			END_IF
		ELSE
			// Set new state command
			eCommand := stModeStateIn.State;
		END_IF

		// Find requested state
		CASE eCommand OF
			E_PML_Command.Reset:
				stModeStateOut.RequestedState := E_PML_State.Idle;

			E_PML_Command.Start:
				stModeStateOut.RequestedState := E_PML_State.Execute;
			
			E_PML_Command.Stop:
				stModeStateOut.RequestedState := E_PML_State.Stopped;
			
			E_PML_Command.Hold:
				stModeStateOut.RequestedState := E_PML_State.Held;
			
			E_PML_Command.Unhold:
				stModeStateOut.RequestedState := E_PML_State.Execute;
			
